      L     #HELP.WZ_rechts_3;
      L     #HELP.WZ_rechts_4;
      +R;
      T     #HELP.Sum_WZ_re_hinten;
      L     #HELP.AW_WZ_re_hinten;
      -R;
      ABS;
      L     #HELP.Tol_UeW_WZ;
      >R;
      A     #OUT.RUECK;
      S     #Kollision;

      A     #Kollision;
      A     #ZST.Unten_re;
      S     #ErrIn.Alarm.Koll_LF;

      A     #Kollision;
      A     #ZST.Oben_re;
      S     #ErrIn.Alarm.Koll_WF;


NETWORK
TITLE = allgemeine Fehlerbehandlung/Überwachungsfunktionen + Fehlerevent
// überwacht die Fahrwagenfunktionen in allen Betriebsarten
// ======== LASER ===========
Err:  L     S5T#5S;
      A     #ZST.AKTIV;
      O     #BA_Wxl;
      SF    T [#Timer3];

      A     T [#Timer3];
      O     #PAR.Free.Laser_req;
      O     "DB_ANLAGE".BA.Mess_on;
      =     #OUT.Req_Laser;

      L     S5T#1M;
      AN    #ZST.Auto;
      SD    T [#Timer0];
      A     "T_Verz_Auto";
      A     T [#Timer0];
      =     #MLD.Warnung.WARN_nAuto;

//--------------------------
//WT am TW nicht umsetzbar (FB9)
//--------------------------
      AN    #ZST.Auto;
      O     #ZST.Halt;
      ON    #ZST.BEREIT;
      O     #IN.QUITT_ALARM;
      O     #F_Taste;
      R     #ErrIn.Warnung.Wrn_WT_nUmsetzbar;

      A     #ErrIn.Warnung.Wrn_WT_nUmsetzbar;
      A     #ZST.Auto;
      =     #MLD.Warnung.WARN_WT_nUms;

//--------------------------
//FW-allgemein
//--------------------------
      A     #ErrIn.Alarm.F_Brk_Fahr;
      =     #MLD.Alarm_HW.F_Brk_Fahr;

//--------------------------
//Positioniersystem
//--------------------------
      AN    #ZST.REFERENZIERT;
      =     #MLD.Alarm_SW.nReferenz;

      A     #ErrIn.Alarm.PosSys;
      =     #MLD.Alarm_HW.PosSys;

      SET;
      R     #ErrPosSys;

      A     #ErrIn.Warnung.Wrn_Optik_PosSys;
      O     #ErrIn.Warnung.Wrn_Temp_PosSys;
      O     #ErrIn.Warnung.Wrn_Plaus_PosSys;
      JC    CNTp;

      L     0;
      T     #HELP.Count_PosSys;
      JU    eRRp;

CNTp: L     #HELP.Count_PosSys;
      L     30;
      >I;
      S     #ErrPosSys;
      JC    eRRp;
      AN    "Imp_1Hz";
      JC    eRRp;
      L     #HELP.Count_PosSys;
      +     1;
      T     #HELP.Count_PosSys;

eRRp: A     #ErrIn.Warnung.Wrn_Optik_PosSys;
      A     #ErrPosSys;
      =     #MLD.Warnung.Optik_PosSys;

      A     #ErrIn.Warnung.Wrn_Temp_PosSys;
      A     #ErrPosSys;
      =     #MLD.Warnung.Temp_PosSys;

      A     #ErrIn.Warnung.Wrn_Plaus_PosSys;
      A     #ErrPosSys;
      =     #MLD.Warnung.Wrn_Plaus_PosSys;

//Einschaltverzögerung Laser
      AN    #OUT.Req_Laser;
      O     #IN.Laser_on;
      L     0;
      JC    Loff;
      L     #HELP.Count_Laser_on;
      AN    "Imp_1Hz";
      JC    Loff;
      +     1;
Loff: T     #HELP.Count_Laser_on;

      L     #HELP.Count_Laser_on;
      L     5;
      >I;
      =     #MLD.Alarm_SW.Laser_off;

      A     #ErrIn.Warnung.Wrn_Temp_Fahr;
      A     #ZST.BEREIT;
      AN    #ErrIn.Alarm.Profinet_IO_nok;
      =     #MLD.Alarm_HW.Temp_Fahrt;
      A     #ErrIn.Warnung.Wrn_Temp_Fahr;
      AN    #ZST.BEREIT;
      AN    #ErrIn.Alarm.Profinet_IO_nok;
      =     #MLD.Warnung.Temp_Fahrt;
      A     #ErrIn.Alarm.Fahrt_nok;
      =     #MLD.Alarm_HW.St_FU_Fahrt;

      A     #ErrIn.Warnung.Wrn_Temp_Hub;
      A     #ZST.BEREIT;
      AN    #ErrIn.Alarm.Profinet_IO_nok;
      =     #MLD.Alarm_HW.Temp_Hub;

      A     #ErrIn.Warnung.Wrn_Temp_Hub;
      AN    #ZST.BEREIT;
      AN    #ErrIn.Alarm.Profinet_IO_nok;
      =     #MLD.Warnung.Temp_Hub;

//--------------------------
//Hubsystem
//--------------------------
      A     #ErrIn.Alarm.HubSys_li;
      =     #MLD.Alarm_HW.HubSys_li;

      A     #ErrIn.Alarm.HubSys_re;
      =     #MLD.Alarm_HW.HubSys_re;

      A     #ErrIn.Alarm.Hub_nok_links;
      =     #MLD.Alarm_HW.St_FU_Hub_li;
      A     #ErrIn.Alarm.Hub_nok_rechts;
      =     #MLD.Alarm_HW.St_FU_Hub_re;

      A     #ErrIn.Alarm.F_Brk_Hub_links;
      =     #MLD.Alarm_HW.F_Brk_Hub_li;
      A     #ErrIn.Alarm.F_Brk_Hub_rechts;
      =     #MLD.Alarm_HW.F_Brk_Hub_re;

//--------------------------
//Bereichs-/Kollisionsfehler
//--------------------------
      A     #ErrIn.Alarm.BE_Vor;
      AN    #ErrIn.Alarm.Profinet_IO_nok;
      =     #MLD.Alarm_HW.BE_vor;
      A     #ErrIn.Alarm.BE_Rck;
      AN    #ErrIn.Alarm.Profinet_IO_nok;
      =     #MLD.Alarm_HW.BE_rck;
      A     #ErrIn.Alarm.Gurt_UP_links;
      AN    #ErrIn.Alarm.Profinet_IO_nok;
      =     #MLD.Alarm_HW.GE_oben_li;
      A     #ErrIn.Alarm.Gurt_DN_links;
      AN    #ErrIn.Alarm.Profinet_IO_nok;
      =     #MLD.Alarm_HW.GE_unten_li;
      A     #ErrIn.Alarm.Gurt_UP_rechts;
      AN    #ErrIn.Alarm.Profinet_IO_nok;
      =     #MLD.Alarm_HW.GE_oben_re;
      A     #ErrIn.Alarm.Gurt_DN_rechts;
      AN    #ErrIn.Alarm.Profinet_IO_nok;
      =     #MLD.Alarm_HW.GE_unten_re;

      A     #ErrIn.Alarm.Koll_LF;
      AN    #ErrIn.Alarm.Profinet_IO_nok;
      S     #MLD.Alarm_HW.Koll_LF;
      A     #ErrIn.Alarm.Koll_WF;
      AN    #ErrIn.Alarm.Profinet_IO_nok;
      S     #MLD.Alarm_HW.Koll_WF;

      A     #ErrIn.Alarm.AFS_BS;
      AN    #ErrIn.Alarm.Profinet_IO_nok;
      =     #MLD.Alarm_HW.Afs_BS;
      A     #ErrIn.Alarm.AFS_WS;
      AN    #ErrIn.Alarm.Profinet_IO_nok;
      =     #MLD.Alarm_HW.Afs_WS;

      A     #ErrIn.Alarm.Last_UeW_links;
      =     #MLD.Alarm_HW.Last_UeW_li;

      A     #ErrIn.Alarm.Last_UeW_rechts;
      =     #MLD.Alarm_HW.Last_UeW_re;

      A     #ErrIn.Alarm.Gurt_UeL_links;
      AN    #ErrIn.Alarm.Profinet_IO_nok;
      =     #MLD.Alarm_HW.GurtUeL_li;

      A     #ErrIn.Alarm.Gurt_UeL_rechts;
      AN    #ErrIn.Alarm.Profinet_IO_nok;
      =     #MLD.Alarm_HW.GurtUeL_re;

      A     #ErrIn.Alarm.Profinet_IO_nok;
      =     #MLD.Alarm_HW.Profinet_nok;

//--------------------------
//Diagnose-/Fehlermeldung
//--------------------------
//:::::::::::::::::::::::::::::::
// Neustart AMS-alle Fehler neu
//:::::::::::::::::::::::::::::::
      AN    "DB_ANLAGE".IN.AMS_Restart;
      JC    NRes;
      L     0;
      T     #MLD.AM_ALHW;
      T     #MLD.AM_ALSW;
      T     #MLD.AM_WARN;
NRes: NOP   0;
//:::::::::::::::::::::::::::::::
// NotAus keine Fehlerbehandlung
//:::::::::::::::::::::::::::::::
      A     #ErrIn.Alarm.NotHalt;
      S     #ZST.FEHLER;
      JC    AOFF;
//:::::::::::::::::::::::::::::::
// Adresse initialisieren
//:::::::::::::::::::::::::::::::
      L     406;
      SLD   3;
      LAR1;
//:::::::::::::::::::::::::::::::
// Schleife über alle Fehler
//:::::::::::::::::::::::::::::::
      L     1;
reA:  T     #TMP.FHLR_NR;
      L     96;
      >I;
      JC    AEnd;
//:::::::::::::::::::::::::::::::
// Fehler gekommen/gegangen
//:::::::::::::::::::::::::::::::
      A     DIX [AR1, P#0.0];
      X     DIX [AR1, P#12.0];
      JCN   nxA;
      A     DIX [AR1, P#0.0];
      =     #new;

AOUT: NOP   0;

//:::::::::::::::::::::::::::::::
// Fehler neu--> Hupe
//:::::::::::::::::::::::::::::::
      A     #new;
      R     "DB_ANLAGE".config.M_Q_Hupe;

//:::::::::::::::::::::::::::::::
// nächster Fehler
//:::::::::::::::::::::::::::::::
nxA:  +AR1  P#0.1;
      L     #TMP.FHLR_NR;
      +     1;
      JU    reA;

//:::::::::::::::::::::::::::::::
// Altmerker Sichern
//:::::::::::::::::::::::::::::::
AEnd: L     %DID406;  //#MLD.Alarm_HW.xx
      T     #MLD.AM_ALHW;
      L     %DID410;  //#MLD.Alarm_SW.xx
      T     #MLD.AM_ALSW;
      L     %DID414;  //#MLD.Warnung.xx
      T     #MLD.AM_WARN;

//:::::::::::::::::::::::::::::::
// Fehlerzustand
//:::::::::::::::::::::::::::::::
      L     #MLD.AM_ALHW;
      L     0;
      <>D;
      O(;
      L     #MLD.AM_ALSW;
      <>D;
      );
      S     #ZST.FEHLER;

//:::::::::::::::::::::::::::::::::
// keine Fehler aber Fehlerzustand
//:::::::::::::::::::::::::::::::::
      L     %DID406;  //#MLD.Alarm_HW.xx
      L     0;
      ==D;
      A(;
      L     %DID410;  //#MLD.Alarm_SW.xx
      ==D;
      );
      A     #ZST.FEHLER;
      AN    #IN.QUITT_ALARM;
      S     #MLD.Alarm_SW.Fehler_Quitt;

      A     #ZST.FEHLER;
      AN    #ZST.Tipp;
      JC    AOFF;

      AN    #ZST.Halt;
      O     #ZST.Tipp;
      JC    WT;

//Alles Aus
AOFF: L     0;  //Ausgänge aus
      T     %DIW68;


NETWORK
TITLE = Warenträgerverwaltung
// kopiert WTs in und aus Positionen
// lädt Parameter usw.
WT:   L     #Adr_IstPos;
      LAR1;
      OPN   "DB_POS";
      L     #PAR.FW_Nr;
      T     DBB [AR1, P#5.0];  //FW_Nr im Bad ungerade
      T     DBB [AR1, P#105.0];  //FW_Nr im Bad gerade

      AN    #WTon_li;
      JC    nUms_li;
      L     #ZST.WT_DB_NR_li;
      +     100;
      T     #WT_DB_NR_li;

      OPN   DB [#WT_DB_NR_li];
      L     #PAR.FW_Nr;
      T     %DBB34;  //"DB_WT1".FW_Nr
nUms_li:A     #WTon_li;
      JC    WTaF_li;
      L     0;
      T     #ZST.Verweil;

WTaF_li:A     #ZST.low_SU_li;
      FN    #TMP.FM_low_SU_li;
      =     #FN_low_SU_li;

      AN    #ZST.Mittig;  //Umladen nur in PosMitte
      JC    WT_rechts;

//--------------------------------
//Kopieren WT in bzw. aus Pos
//--------------------------------
      A     #ZST.low_SU_li;
      A     #WTon_li;
      AN    #WT_in_Pos_li;
      A     #TMP.old_hub;  //#ZST.SENKEN_AKT
      JC    WT_P_li;
      A     #FN_low_SU_li;
      AN    #WTon_li;
      A     #WT_in_Pos_li;
      A     #TMP.old_hub;  //#ZST.HEBEN_AKT
      JC    WT_F_li;
      JU    WT_rechts;
//--------------------------------
//WT in Position laden
//--------------------------------
WT_P_li:L     #ZST.POSITION_li;
      T     #Nummer;

      CALL  "FC_WT_to_Pos"
      ( Pos_Nr     := #Nummer,
        WT_Nr      := #ZST.WT_DB_NR_li,
        BA_Auto    := #ZST.Auto,
        send_DBEvt := TRUE,
        SimLoad    := FALSE,
        Copy_ok    := #"Return"
      );

      AN    #"Return";
      JC    WT_rechts;
      R     #WTon_li;

      L     0;  //löschen am FW
      T     #ZST.WT_DB_NR_li;
      T     #ZST.WT_NR_LANG_li;
      JU    WT_rechts;

//--------------------------------
//WT aus Position laden
//--------------------------------
WT_F_li:L     #ZST.POSITION_li;
      T     #Nummer;

      CALL  "FC_WT_from_Pos"
      ( Pos_Nr     := #Nummer,
        send_DBEvt := TRUE,
        load_ok    := #"Return",
        WT_Nr      := #ZST.WT_DB_NR_li,
        WT_Nr_lang := #ZST.WT_NR_LANG_li
      );

      AN    #"Return";
      JC    WT_rechts;
      S     #WTon_li;

      AN    #ZST.Auto;
      JC    WT_rechts;

      L     #ZST.WT_DB_NR_li;
      +     100;
      T     #WT_DB_NR_li;

      OPN   DB [#WT_DB_NR_li];
      L     %DBB36;  //WT-Ziel bereits festgelegt
      L     0;
      <>I;
      JC    Zset_li;
      L     %DBB21;
      T     %DBB36;  //WT-Ziel

Zset_li:L     #TMP.ZielPos;
      T     %DBB21;

      L     #TMP.ZielPos;
      T     #Nummer;
      CALL  "FC_WT_to_Pos"
      ( Pos_Nr     := #Nummer,
        WT_Nr      := #ZST.WT_DB_NR_li,
        BA_Auto    := #ZST.Auto,
        send_DBEvt := FALSE,
        SimLoad    := TRUE,
        Copy_ok    := #"Return"
      );

WT_rechts:NOP   0;

      AN    #WTon_re;
      JC    nUms_re;
      L     #ZST.WT_DB_NR_re;
      +     100;
      T     #WT_DB_NR_re;

      OPN   DB [#WT_DB_NR_re];
      L     #PAR.FW_Nr;
      T     %DBB34;  //"DB_WT1".FW_Nr
nUms_re:A     #WTon_re;
      JC    WTaF_re;
      L     0;
      T     #ZST.Verweil;

WTaF_re:A     #ZST.low_SU_re;
      FN    #TMP.FM_low_SU_re;
      =     #FN_low_SU_re;

      AN    #ZST.Mittig;  //Umladen nur in PosMitte
      JC    Komm;

//--------------------------------
//Kopieren WT in bzw. aus Pos
//--------------------------------
      A     #ZST.low_SU_re;
      A     #WTon_re;
      AN    #WT_in_Pos_re;
      A     #TMP.old_hub;  //#ZST.SENKEN_AKT
      JC    WT_P_re;
      A     #FN_low_SU_re;
      AN    #WTon_re;
      A     #WT_in_Pos_re;
      A     #TMP.old_hub;  //#ZST.HEBEN_AKT
      JC    WT_F_re;
      JU    Komm;
//--------------------------------
//WT in Position laden
//--------------------------------
WT_P_re:L     #ZST.POSITION_re;
      T     #Nummer;

      CALL  "FC_WT_to_Pos"
      ( Pos_Nr     := #Nummer,
        WT_Nr      := #ZST.WT_DB_NR_re,
        BA_Auto    := #ZST.Auto,
        send_DBEvt := TRUE,
        SimLoad    := FALSE,
        Copy_ok    := #"Return"
      );

      AN    #"Return";
      JC    Komm;
      R     #WTon_re;

      L     0;  //löschen am FW
      T     #ZST.WT_DB_NR_re;
      T     #HELP.WT_NR_LANG_re;
      JU    Komm;

//--------------------------------
//WT aus Position laden
//--------------------------------
WT_F_re:L     #ZST.POSITION_re;
      T     #Nummer;

      CALL  "FC_WT_from_Pos"
      ( Pos_Nr     := #Nummer,
        send_DBEvt := TRUE,
        load_ok    := #"Return",
        WT_Nr      := #ZST.WT_DB_NR_re,
        WT_Nr_lang := #HELP.WT_NR_LANG_re
      );

      AN    #"Return";
      JC    Komm;
      S     #WTon_re;

      AN    #ZST.Auto;
      JC    Komm;

      L     #ZST.WT_DB_NR_re;
      +     100;
      T     #WT_DB_NR_re;

      OPN   DB [#WT_DB_NR_re];
      L     %DBB36;  //WT-Ziel bereits festgelegt
      L     0;
      <>I;
      JC    Zset_re;
      L     %DBB21;
      T     %DBB36;  //WT-Ziel

Zset_re:L     #TMP.ZielPos;
      T     %DBB21;

      L     #TMP.ZielPos;
      T     #Nummer;
      CALL  "FC_WT_to_Pos"
      ( Pos_Nr     := #Nummer,
        WT_Nr      := #ZST.WT_DB_NR_re,
        BA_Auto    := #ZST.Auto,
        send_DBEvt := FALSE,
        SimLoad    := TRUE,
        Copy_ok    := #"Return"
      );


NETWORK
TITLE = Kommunikation zu Partnerfunktionen
// Datenübertragung zu PC, Optimierung, Diagwatch usw.
// Ziel-Quelle-Informationen, Heben-Senken-Informationen in Positionen anmelden
Komm: NOP   0;
//---------------------------
//Positionsinformationen DB51
//---------------------------
      L     #Adr_IstPos;
      LAR1;
      OPN   "DB_POS";
      A     #ZST.HEBEN_AKT;  // #OUT.HEBEN
      =     DBX [AR1, P#6.6];  //FW Heben
      =     DBX [AR1, P#106.6];  //FW Heben
      A     #ZST.SENKEN_AKT;  // #OUT.SENKEN
      =     DBX [AR1, P#6.7];  //FW Senken
      =     DBX [AR1, P#106.7];  //FW Senken

      AN    #ZST.VORWAERTS_AKT;
      AN    #ZST.RUECKWAERTS_AKT;
      A     #ZST.Mittig;
      =     DBX [AR1, P#6.5];  //FW in Pos
      =     DBX [AR1, P#106.5];  //FW in Pos

//FW-kommt in allen Positionen setzen,die überfahren werden
      L     0;
      L     #TMP.ZielPos;
      ==I;
      JC    noZ;
      L     2;
      MOD;
      L     #TMP.ZielPos;
      JP    linke_S;
      DEC   1;
linke_S:L     #ZST.POSITION_li;
      <I;
      JC    ldC;
      CAC;
ldC:  T     #PCount_hi;
      CAC;
retC: T     #PCount_low;
      L     "DB_POS".LENG;
      *I;
      L     "DB_POS".Offset;
      +I;
      SLD   3;
      LAR1;
      OPN   "DB_POS";
      S     DBX [AR1, P#6.4];  //FW kommt
      S     DBX [AR1, P#106.4];  //FW kommt
      L     #PCount_hi;
      L     #PCount_low;
      <=I;
      JC    noZ;
      +     2;
      JU    retC;

noZ:  AN    #ZST.Auto;
      JC    noto;
      L     %DIB31;  //Befehlsart
      L     16#03;
      <>I;
      JC    noto;
//Ziel sperren
      L     0;
      L     %DIB33;
      ==I;
      JC    noto;
      L     "DB_POS".LENG;
      *I;
      L     "DB_POS".Offset;
      +I;
      SLD   3;
      LAR1;
      OPN   "DB_POS";
      S     DBX [AR1, P#6.3];  //reserviertes Ziel
      AN    #WTon_li;
      AN    #WTon_re;
      JC    Qset;

      AN    #WTon_li;
      JC    rZ_re;
      L     #ZST.WT_DB_NR_li;
      T     DBB [AR1, P#36.0];  //Next-WT

      AN    #WTon_re;
      JC    Qset;
      L     #ZST.WT_DB_NR_re;
      T     DBB [AR1, P#136.0];  //Next-WT
      JU    Qset;

rZ_re:AN    #WTon_re;
      JC    Qset;
      L     #ZST.WT_DB_NR_re;
      T     DBB [AR1, P#36.0];  //Next-WT

//Quelle sperren
Qset: A     #WTon_li;
      O     #WTon_re;
      JC    noto;
      L     0;
      L     %DIB32;
      ==I;
      JC    noto;
      L     "DB_POS".LENG;
      *I;
      L     "DB_POS".Offset;
      +I;
      SLD   3;
      LAR1;
      OPN   "DB_POS";
      S     DBX [AR1, P#6.2];  //reservierte Quelle

noto: BE;

END_FUNCTION_BLOCK

FUNCTION "FC_Pos_Erk" : Void   // FC11, STL
TITLE = Positioniersystem
{ S7_Optimized_Access := 'FALSE' }
AUTHOR : MS
FAMILY : FW
// stored: AutoNumber false
   VAR_INPUT
      Instanz_DB : Int;
   END_VAR
   VAR_TEMP
      FW_DB : DB_ANY;
      Abstand : DInt;
      Pos : Byte;
      count : Byte;
      rotWert : Word;
      frstChk : Bool;
      minGrenze : Byte;
      maxGrenze : Byte;
      Grenze_min : DInt;
      Grenze_max : DInt;
      SU_Ebene_0 : DInt;
   END_VAR
BEGIN

NETWORK
TITLE = Position ermitteln
// Inkrementwert wird auf minimalen Abstand einer Positionsmitte überprüft.
// Position mit geringstem Abstand wird übernommen.
      L     #Instanz_DB;
      T     #FW_DB;
      OPN   DI [#FW_DB];

      SET;
      =     #frstChk;
      L     0;
      T     #SU_Ebene_0;

      L     "DI_FW_1".PAR.Fahrt.FAHRBEREICH_MIN;
      T     #minGrenze;
      L     "DI_FW_1".PAR.Fahrt.FAHRBEREICH_MAX;
      T     #maxGrenze;
      L     "DI_FW_1".IN.Grenze_min;
      T     #Grenze_min;
      L     "DI_FW_1".IN.Grenze_max;
      T     #Grenze_max;

      L     "DI_FW_1".PAR.Fahrt.FAHRBEREICH_MIN;
      T     #Pos;
retP: T     #count;
      L     "DI_FW_1".PAR.Fahrt.FAHRBEREICH_MAX;
      +     -1;  // HCA: nur ungerade Pos. zählen
      >I;
      JC    ckok;

      L     #count;
      L     "DB_POS".LENG;
      *D;
      L     "DB_POS".Offset;
      +D;
      SLD   3;
      LAR1;
      OPN   "DB_POS";
      L     #Grenze_min;
      L     DBD [AR1, P#22.0];  //BadPos in Inc
      <=D;
      JC    gmin;
      L     #count;
      +     2;  // HCA: nur ungeradePos. zählen
      T     #minGrenze;
gmin: L     #Grenze_max;
      OPN   "DB_POS";
      L     DBD [AR1, P#22.0];  //BadPos in Inc
      <D;
      JC    gmax;
      L     #count;
      T     #maxGrenze;
gmax: NOP   0;
      OPN   "DB_POS";
      L     DBD [AR1, P#22.0];  //BadPos in Inc
      L     "DI_FW_1".ZST.PosInc;
      -D;
      DTR;
      ABS;
      RND;
      L     #Abstand;
      >=D;
      AN    #frstChk;
      JC    nexP;
      R     #frstChk;
      CAC;
      T     #Abstand;
      L     #count;
      T     #Pos;

nexP: L     #count;
      L     2;  // HCA: nur ungeradePos. zählen
      +I;
      JU    retP;

ckok: L     #Pos;
      T     "DI_FW_1".ZST.POSITION_li;

      L     #Abstand;
      L     "DI_FW_1".PAR.Fahrt.Bereich_Pos;
      <=D;
      =     "DI_FW_1".ZST.Mittig;

// Ofs-Mittig
      L     #Pos;
      L     "DB_POS".LENG;
      *D;
      L     "DB_POS".Offset;
      +D;
      SLD   3;
      LAR1;
      OPN   "DB_POS";
      L     DBD [AR1, P#22.0];  //BadPos in Inc
      L     DBD [AR1, P#64.0];  //"DB_POS".POS[x].SonderPos_Offset
      -D;
      L     "DI_FW_1".ZST.PosInc;
      -D;
      DTR;
      ABS;
      RND;
      L     "DI_FW_1".PAR.Fahrt.Bereich_Pos;
      <=D;
      =     "DI_FW_1".ZST.Ofs_mittig;

// Tiefsenkbereich
      A(;
      OPN   "DB_POS";
      L     DBD [AR1, P#22.0];  //Posmitte
      L     "DI_FW_1".PAR.Fahrt.Bereich_Pos;
      +D;
      L     "DI_FW_1".ZST.PosInc;
      >D;
      );
      A(;
      OPN   "DB_POS";
      L     DBD [AR1, P#22.0];  //Posmitte
      L     DBD [AR1, P#64.0];  //"DB_POS".POS[x].SonderPos_Offset
      -D;
      L     "DI_FW_1".PAR.Fahrt.Bereich_Pos;
      -D;
      L     "DI_FW_1".ZST.PosInc;
      <D;
      );
      A(;
      A     "DI_FW_1".IN.Unten_li;
      O     "DI_FW_1".IN.Unten_re;
      );
      =     "DI_FW_1".ZST.Ofs_Bereich;

// Absetzhöhe
      OPN   "DB_POS";
      L     0;
      L     DBD [AR1, P#14.0];  //"DB_POS".POS[x].Absetzhoehe
      >=D;
      JC    VZB;
      T     "DI_FW_1".PAR.Hub.Ebene0;

//Vorzugsbereich min ungültig?
VZB:  L     "DI_FW_1".PAR.Fahrt.FAHRBEREICH_MIN;
      L     "DI_FW_1".PAR.Vorzugsbereich_max;
      >I;
      O(;
      L     "DI_FW_1".PAR.Fahrt.FAHRBEREICH_MAX;
      >I;
      );
      JC    Gclr;
//ggf. Korrektur min
      L     #maxGrenze;
      L     "DI_FW_1".PAR.Vorzugsbereich_max;
      <=I;
      JC    Gclr;
      T     #minGrenze;
Gclr: NOP   0;

//Vorzugsbereich min ungültig?
      L     "DI_FW_1".PAR.Fahrt.FAHRBEREICH_MIN;
      L     "DI_FW_1".PAR.Vorzugsbereich_min;
      >I;
      O(;
      L     "DI_FW_1".PAR.Fahrt.FAHRBEREICH_MAX;
      >I;
      );
      JC    Gset;
//ggf. Korrektur min
      L     #minGrenze;
      L     "DI_FW_1".PAR.Vorzugsbereich_min;
      >=I;
      JC    Gset;
      T     #minGrenze;

Gset: L     #minGrenze;
      T     "DI_FW_1".HELP.Grenze_min;
      L     #maxGrenze;
      T     "DI_FW_1".HELP.Grenze_max;




NETWORK
TITLE = nächsten HW ermitteln
ChHW: NOP   0;
      AN    "DB_ANLAGE".config.HW_exist;
      R     "DI_FW_1".ZST.HW_mittig;
      L     1;  //temp. Hubeben
      JC    SUok;

      SET;
      =     #frstChk;

      L     0;
      T     #Pos;
retH: T     #count;
      L     "DB_HW".Anzahl;
      >=I;
      JC    Hok;

      L     #count;
      L     "DB_HW".lengHW;
      *D;
      L     "DB_HW".Offset;
      +D;
      SLD   3;
      LAR1;
      OPN   "DB_HW";
      L     0;
      L     DBD [AR1, P#0.0];  //HW-Pos in Inc
      ==D;
      JC    Hok;
      L     "DI_FW_1".ZST.PosInc;
      -D;
      DTR;
      ABS;
      RND;
      L     #Abstand;
      >=D;
      AN    #frstChk;
      JC    nexH;
      R     #frstChk;
      CAC;
      T     #Abstand;
      L     #count;
      T     #Pos;

nexH: L     #count;
      L     1;
      +I;
      JU    retH;

Hok:  L     #Abstand;
      L     "DI_FW_1".PAR.Fahrt.Bereich_Pos;
      <=D;
      =     "DI_FW_1".ZST.HW_mittig;


NETWORK
TITLE = aktuelle SU-Ebene ermitteln
      L     #Pos;
      L     "DB_HW".lengHW;
      *D;
      L     "DB_HW".Offset;
      +D;
      SLD   3;
      LAR1;
      A     "DI_FW_1".ZST.HW_mittig;
      JC    mitt;
      OPN   "DB_HW";
      L     DBD [AR1, P#0.0];  //HW-Pos in Inc
      L     "DI_FW_1".ZST.PosInc;
      -D;
      JP    vorH;
//FW ist hinter HW-Pos
      OPN   "DB_HW";
      L     DBB [AR1, P#5.0];  //HW-Ebene bei verlassen in Richtung vorwärts
      T     "DI_FW_1".TMP.low_SU_Ebene;
      L     1;
      SLW;  //Bit0==TRUE wird um Ebene verschoben
      JU    SUok;

//FW ist vor HW-Pos
vorH: OPN   "DB_HW";
      L     DBB [AR1, P#4.0];  //HW-Ebene bei verlassen in Richtung rückwärts
      T     "DI_FW_1".TMP.low_SU_Ebene;
      L     1;
      SLW;  //Bit0==TRUE wird um Ebene verschoben
      JU    SUok;

//FW ist auf HW-Pos
mitt: OPN   "DB_HW";
      L     DBB [AR1, P#4.0];  //HW-Ebene bei verlassen in Richtung rückwärts
      L     DBB [AR1, P#5.0];  //HW-Ebene bei verlassen in Richtung vorwärts
      >I;
      JC    lSU;
      CAC;
lSU:  T     "DI_FW_1".TMP.low_SU_Ebene;
      OPN   "DB_HW";
      L     DBB [AR1, P#4.0];  //HW-Ebene bei verlassen in Richtung rückwärts
      L     1;
      SLW;  //Bit0==TRUE wird um Ebene verschoben
      T     #rotWert;
      L     DBB [AR1, P#5.0];  //HW-Ebene bei verlassen in Richtung vorwärts
      L     1;
      SLW;  //Bit0==TRUE wird um Ebene verschoben
      L     #rotWert;
      OW;  //beide Ebenen gelten

SUok: T     "DI_FW_1".TMP.Hub_Ebenen;

      L     "DI_FW_1".TMP.low_SU_Ebene;
      T     "DI_FW_1".PAR.Hub.SUF_Ebene;

      A     "DI_FW_1".ZST.Mittig;
      O     "DI_FW_1".ZST.Ofs_Bereich;
      O     "DI_FW_1".ZST.Ofs_mittig;
      JCN   Z_E;
      L     0;
      T     "DI_FW_1".TMP.low_SU_Ebene;  // ganz unten erlaubt
      L     "DI_FW_1".TMP.Hub_Ebenen;
      OW    W#16#01;
      T     "DI_FW_1".TMP.Hub_Ebenen;

//SO- und Z-Ebene übergeben
Z_E:  L     0;
      L     "DI_FW_1".PAR.Hub.Z_Ebene;
      ==I;
      JC    SO;
      L     1;
      SLW;
      L     "DI_FW_1".TMP.Hub_Ebenen;
      OW;
      T     "DI_FW_1".TMP.Hub_Ebenen;
SO:   L     0;
      L     "DI_FW_1".PAR.Hub.SO_Ebene;
      ==I;
      BEC;
      L     1;
      SLW;
      L     "DI_FW_1".TMP.Hub_Ebenen;
      OW;
      T     "DI_FW_1".TMP.Hub_Ebenen;

END_FUNCTION

FUNCTION "FC_Hub_Erk_li" : Void   // FC12, STL
TITLE = Hubsystem
{ S7_Optimized_Access := 'FALSE' }
AUTHOR : MS
FAMILY : FW
// stored: AutoNumber false
   VAR_INPUT
      Instanz_DB : Int;
   END_VAR
   VAR_TEMP
      FW_DB : DB_ANY;
      Abstand : DInt;
      Ebene : Byte;
      count : Byte;
      rotWert : Word;
      frstChk : Bool;
   END_VAR
BEGIN

NETWORK
TITLE = Fahrwagen-Ebene ermitteln
// Inkrementwert wird auf minimalen Abstand zu einer Hubebene überprüft.
// Ebene mit geringstem Abstand wird übernommen.
      L     #Instanz_DB;
      T     #FW_DB;
      OPN   DI [#FW_DB];

      SET;
      =     #frstChk;

      L     0;
      T     #Ebene;
      T     #Abstand;
retE: T     #count;
      L     6;
      >I;
      JC    ckok;

      CAC;
      L     4;
      *D;
      L     292;
      +D;
      SLD   3;
      LAR1;

      L     0;
      L     DID [AR1, P#0.0];  //"DI_FW_1".PAR.Hub.Ebene...
      ==D;
      JC    ckok;
      L     "DI_FW_1".ZST.HubInc_li;
      -D;
      DTR;
      ABS;
      RND;
      L     #Abstand;
      >=D;
      AN    #frstChk;
      JC    nexE;
      R     #frstChk;
      CAC;
      T     #Abstand;
      L     #count;
      T     #Ebene;

nexE: L     #count;
      L     1;
      +I;
      JU    retE;

ckok: L     320;  //prüfen auf Z-Ebene
      SLD   3;
      LAR1;
      L     0;
      L     DID [AR1, P#0.0];  //"DI_FW_1".PAR.Hub.Ebene...
      ==D;
      JC    noZ;
      L     "DI_FW_1".ZST.HubInc_li;
      -D;
      DTR;
      ABS;
      RND;
      L     #Abstand;
      >=D;
      JC    noZ;
      CAC;
      T     #Abstand;
      L     7;
      T     #Ebene;

noZ:  L     #Ebene;
      T     "DI_FW_1".ZST.Ebene_li;

      L     #Abstand;
      L     "DI_FW_1".PAR.Hub.Bereich_Pos;
      <=D;
      AN    #frstChk;
      =     "DI_FW_1".ZST.HubSensor_li;


NETWORK
TITLE = SU/SO/Z setzen

      L     #Ebene;
      L     1;
      SLW;
      L     "DI_FW_1".PAR.Hub.SU_Ebenen;
      AW;
      L     "DI_FW_1".TMP.Hub_Ebenen;
      AW;
      L     0;
      <>I;
      A     "DI_FW_1".ZST.HubSensor_li;
      =     "DI_FW_1".ZST.Unten_li;

      L     #Ebene;
      L     "DI_FW_1".PAR.Hub.Z_Ebene;
      ==I;
      A     "DI_FW_1".ZST.HubSensor_li;
      =     "DI_FW_1".ZST.Z_Sensor_li;

      L     #Ebene;
      L     "DI_FW_1".PAR.Hub.SO_Ebene;
      ==I;
      A     "DI_FW_1".ZST.HubSensor_li;
      =     "DI_FW_1".ZST.Oben_li;

      L     #Ebene;
      L     0;
      ==I;
      R     "DI_FW_1".ZST.Z_Sensor_li;
      R     "DI_FW_1".ZST.Oben_li;

      A     "DI_FW_1".IN.Oben_li;
      S     "DI_FW_1".ZST.Oben_li;


NETWORK
TITLE = WT Kopierfreigabe
      L     "DI_FW_1".TMP.low_SU_Ebene;
      L     #Ebene;
      ==I;
      A     "DI_FW_1".ZST.HubSensor_li;
      =     "DI_FW_1".ZST.low_SU_li;

END_FUNCTION

FUNCTION "FC_Hub_Erk_re" : Void   // FC112, STL
TITLE = Hubsystem
{ S7_Optimized_Access := 'FALSE' }
AUTHOR : MS
FAMILY : FW
// stored: AutoNumber false
   VAR_INPUT
      Instanz_DB : Int;
   END_VAR
   VAR_TEMP
      FW_DB : DB_ANY;
      Abstand : DInt;
      Ebene : Byte;
      count : Byte;
      rotWert : Word;
      frstChk : Bool;
   END_VAR
BEGIN

NETWORK
TITLE = Fahrwagen-Ebene ermitteln
// Inkrementwert wird auf minimalen Abstand zu einer Hubebene überprüft.
// Ebene mit geringstem Abstand wird übernommen.
      L     #Instanz_DB;
      T     #FW_DB;
      OPN   DI [#FW_DB];

      SET;
      =     #frstChk;

      L     0;
      T     #Ebene;
      T     #Abstand;
retE: T     #count;
      L     6;
      >I;
      JC    ckok;

      CAC;
      L     4;
      *D;
      L     292;
      +D;
      SLD   3;
      LAR1;

      L     0;
      L     DID [AR1, P#0.0];  //"DI_FW_1".PAR.Hub.Ebene...
      ==D;
      JC    ckok;
      L     "DI_FW_1".HELP.HubInc_re;
      -D;
      DTR;
      ABS;
      RND;
      L     #Abstand;
      >=D;
      AN    #frstChk;
      JC    nexE;
      R     #frstChk;
      CAC;
      T     #Abstand;
      L     #count;
      T     #Ebene;

nexE: L     #count;
      L     1;
      +I;
      JU    retE;

ckok: L     320;  //prüfen auf Z-Ebene
      SLD   3;
      LAR1;
      L     0;
      L     DID [AR1, P#0.0];  //"DI_FW_1".PAR.Hub.Ebene...
      ==D;
      JC    noZ;
      L     "DI_FW_1".HELP.HubInc_re;
      -D;
      DTR;
      ABS;
      RND;
      L     #Abstand;
      >=D;
      JC    noZ;
      CAC;
      T     #Abstand;
      L     7;
      T     #Ebene;

noZ:  L     #Ebene;
      T     "DI_FW_1".ZST.Ebene_re;

      L     #Abstand;
      L     "DI_FW_1".PAR.Hub.Bereich_Pos;
      <=D;
      AN    #frstChk;
      =     "DI_FW_1".ZST.HubSensor_re;


NETWORK
TITLE = SU/SO/Z setzen

      L     #Ebene;
      L     1;
      SLW;
      L     "DI_FW_1".PAR.Hub.SU_Ebenen;
      AW;
      L     "DI_FW_1".TMP.Hub_Ebenen;
      AW;
      L     0;
      <>I;
      A     "DI_FW_1".ZST.HubSensor_re;
      =     "DI_FW_1".ZST.Unten_re;

      L     #Ebene;
      L     "DI_FW_1".PAR.Hub.Z_Ebene;
      ==I;
      A     "DI_FW_1".ZST.HubSensor_re;
      =     "DI_FW_1".ZST.Z_Sensor_re;

      L     #Ebene;
      L     "DI_FW_1".PAR.Hub.SO_Ebene;
      ==I;
      A     "DI_FW_1".ZST.HubSensor_re;
      =     "DI_FW_1".ZST.Oben_re;

      L     #Ebene;
      L     0;
      ==I;
      R     "DI_FW_1".ZST.Z_Sensor_re;
      R     "DI_FW_1".ZST.Oben_re;

      A     "DI_FW_1".IN.Oben_re;
      S     "DI_FW_1".ZST.Oben_re;


NETWORK
TITLE = WT Kopierfreigabe
      L     "DI_FW_1".TMP.low_SU_Ebene;
      L     #Ebene;
      ==I;
      A     "DI_FW_1".ZST.HubSensor_re;
      =     "DI_FW_1".ZST.low_SU_re;

END_FUNCTION

FUNCTION "FC_Transzeit" : Void   // FC35, STL
{ S7_Optimized_Access := 'FALSE' }
AUTHOR : MS
// stored: AutoNumber false
   VAR_INPUT
      Pos : Byte;
      Quelle : Byte;
      Ziel : Byte;
      FW_Nr : Byte;
      ChkLeerfahrt : Bool;   // nur Leerfahrt berechnen
      StartPos : Bool;   // inc. der Pos als Startposition
      KorrTime : DInt;   // Korrektur Zeit in der Zukunft
   END_VAR
   VAR_OUTPUT
      Fahrzeit : DInt;
   END_VAR
   VAR_TEMP
      Leerfahrt : Real;
      Hubzeit : Real;
      Tropfzeit : Real;
      Warenfahrt : Real;
      Pendelzeit : Real;
      Senkzeit : Real;
      Tropfwanne : Real;
      KorrAtz : Real;
      KorrPend : Real;
      Trommel : Bool;
      lngsm_h : Bool;
      lngsm_s : Bool;
      FWok : Bool;
      immer_schnell : Bool;
      TS_Pos : Bool;
      WT_DB : Int;
      savAr1 : DWord;
      FW_DB : Int;
      Abstand : Real;
      ProzSpeed : Real;
      Quellpos : DInt;
      Restzeit : DInt;
      IstInc : DInt;
   END_VAR
BEGIN

NETWORK
TITLE = Register retten
// --------------------------------
// Register retten
// --------------------------------
      TAR1;
      T     #savAr1;


NETWORK
TITLE = Init
      L     0;
      T     #Fahrzeit;
      T     #Leerfahrt;
      T     #Hubzeit;
      T     #Tropfzeit;
      T     #Warenfahrt;
      T     #Pendelzeit;
      T     #Senkzeit;
      T     #Tropfwanne;

      SET;
      =     #TS_Pos;

      L     #FW_Nr;
      L     0;
      >I;
      =     #FWok;

      L     #FW_Nr;
      L     "DB_ANLAGE".config.ANZ_FW;
      >I;
      R     #FWok;
      R     #TS_Pos;

      L     1;
      L     #Quelle;
      >I;
      O(;
      L     "DB_ANLAGE".config.ANZ_Pos;
      >I;
      );
      JC    raus;

      A     #ChkLeerfahrt;
      JC    Leer;

      L     1;
      L     #Ziel;
      >I;
      O(;
      L     "DB_ANLAGE".config.ANZ_Pos;
      >I;
      );
      JC    raus;

Leer: NOP   0;

NETWORK
TITLE = Leerfahrt
      L     #Pos;
      L     "DB_POS".LENG;
      *D;
      L     "DB_POS".Offset;
      +D;
      SLD   3;
      LAR1;
      OPN   "DB_POS";
      L     DBD [AR1, P#22.0];  //"DB_POS".POS[0].IncPos
      T     #IstInc;

      L     #Quelle;
      L     "DB_POS".LENG;
      *D;
      L     "DB_POS".Offset;
      +D;
      SLD   3;
      LAR1;
      OPN   "DB_POS";
      AN    DBX [AR1, P#8.0];  //"DB_POS".POS[0].TS_Pos
      R     #TS_Pos;
      A     DBX [AR1, P#10.2];  //"DB_POS".POS[0].ignor_Exp
      L     0;
      JC    okRT;
      L     DBD [AR1, P#60.0];  //"DB_POS".POS[0].Korr_Restzeit
      L     #KorrTime;
      -D;
      JP    okRT;
      L     0;
okRT: DTR;
      T     #Restzeit;

      A     #FWok;
      A     "DB_ANLAGE".config.Pos_absolut;
      JC    LFa;

//Leerfahrzeit Sensor berechnen
      L     #Pos;
      L     #Quelle;
      -I;
      ITD;
      DTR;
      ABS;
      L     0.0;
      ==R;
      JC    LF;
      CAC;
      L     1.0;
      -R;
      L     "DB_Fahr-Hubzeit".FZ_Typ_Pos;
      *R;
      L     "DB_Fahr-Hubzeit".FZ_Typ_Halt;
      +R;
      JU    LF;

//Leerfahrzeit absolut berechnen
LFa:  L     #Quelle;
      L     "DB_POS".LENG;
      *D;
      L     "DB_POS".Offset;
      +D;
      SLD   3;
      LAR1;
      OPN   "DB_POS";
      L     DBD [AR1, P#22.0];  //"DB_POS".POS[0].IncPos
      T     #Quellpos;
      L     DBB [AR1, P#36.0];  //WT-DB
      +     100;
      T     #WT_DB;

      L     #FW_Nr;
      +     10;
      T     #FW_DB;

      A     #StartPos;
      L     #IstInc;
      JC    EPQ;

      OPN   DB [#FW_DB];
      L     0;
      L     %DBW366;  //"DI_FW_1".TMP.EndZiel
      ==I;
      JC    rdyQ;
      L     "DB_POS".LENG;
      *D;
      L     "DB_POS".Offset;
      +D;
      SLD   3;
      LAR1;
      OPN   "DB_POS";
      L     DBD [AR1, P#22.0];  //"DB_POS".POS[0].IncPos
      JU    EPQ;

rdyQ: OPN   DB [#FW_DB];
      L     %DBD4;  //"DI_FW_1".ZST.PosInc
EPQ:  L     #Quellpos;
      -D;
      DTR;
      ABS;
      T     #Abstand;
      L     0.0;
      ==D;
      JC    LF;

      OPN   DB [#FW_DB];
      L     %DBW246;  //"DI_FW_1".PAR.Fahrt.Fahr_DBNr
      T     #FW_DB;
      OPN   DB [#FW_DB];
      L     %DBW12;  //"DI_FW_POS_1".Config.Speed.Max
      ITD;
      DTR;
      L     100.0;
      /R;
      T     #ProzSpeed;

      L     %DBD22;  //"DI_FW_POS_1".Config.Rampe.Auf_Leer
      L     %DBD26;  //"DI_FW_POS_1".Config.Rampe.Ab_Leer
      +R;
      L     2.0;
      /R;
      L     #ProzSpeed;
      *R;
      T     #Leerfahrt;  //Zeit für Rampen
      L     %DBD14;  //"DI_FW_POS_1".Config.Speed.Norm mm/s
      *R;
      L     2.0;
      /R;
      L     #Abstand;
      CAC;
      -R;
      T     #Abstand;  //Weg für Konstantfahrt
      L     0.0;
      <=R;
      JC    endL;

      L     %DBD14;  //"DI_FW_POS_1".Config.Speed.Norm mm/s
      L     #ProzSpeed;
      *R;
      L     #Abstand;
      CAC;
      /R;
      L     #Leerfahrt;
      +R;
LF:   T     #Leerfahrt;
endL: SET;
      A     #ChkLeerfahrt;
      JC    Zeit;

NETWORK
TITLE = Warenfahrt
      L     #Quelle;
      L     #Ziel;
      -I;
      ITD;
      DTR;
      ABS;
      L     0.0;
      ==R;
      JC    WF;

      A     #FWok;
      A     "DB_ANLAGE".config.Pos_absolut;
      JC    WFa;
//Warenfahrzeit Sensor berechnen
      CAC;
      L     1.0;
      -R;
      L     "DB_Fahr-Hubzeit".FZ_Typ_Pos;
      *R;
      L     "DB_Fahr-Hubzeit".FZ_Typ_Halt;
      +R;
      JU    WF;

//Warenfahrzeit absolut berechnen
WFa:  L     #Ziel;
      L     "DB_POS".LENG;
      *D;
      L     "DB_POS".Offset;
      +D;
      SLD   3;
      LAR1;
      OPN   "DB_POS";
      L     DBD [AR1, P#22.0];  //"DB_POS".POS[0].IncPos
      L     #Quellpos;
      -D;
      DTR;
      ABS;
      T     #Abstand;
      L     0.0;
      ==D;
      JC    WF;

      L     1.0;
      T     #ProzSpeed;

      L     100;
      L     #WT_DB;
      >=I;
      JC    nWT;
      OPN   DB [#WT_DB];
      L     %DBW68;  //"DB_WT1".Speed_Fahrt
      ITD;
      DTR;
      L     100.0;
      /R;
      T     #ProzSpeed;

nWT:  L     #FW_Nr;
      +     10;
      T     #FW_DB;

      OPN   DB [#FW_DB];
      AN    %DBX343.0;  //"DI_FW_1".PAR.Free.TS
      R     #TS_Pos;
      L     %DBW246;  //"DI_FW_1".PAR.Fahrt.Fahr_DBNr
      T     #FW_DB;
      OPN   DB [#FW_DB];
      L     %DBW12;  //"DI_FW_POS_1".Config.Speed.Max
      ITD;
      DTR;
      L     100.0;
      /R;
      L     #ProzSpeed;
      *R;
      T     #ProzSpeed;

      L     %DBD30;  //"DI_FW_POS_1".Config.Rampe.Auf_Ware
      L     %DBD34;  //"DI_FW_POS_1".Config.Rampe.Ab_Ware
      +R;
      L     2.0;
      /R;
      L     #ProzSpeed;
      *R;
      T     #Warenfahrt;  //Zeit für Rampen
      L     %DBD14;  //"DI_FW_POS_1".Config.Speed.Norm mm/s
      *R;
      L     2.0;
      /R;
      L     #Abstand;
      CAC;
      -R;
      T     #Abstand;  //Weg für Konstantfahrt
      L     0.0;
      <=R;
      JC    endW;

      L     %DBD14;  //"DI_FW_POS_1".Config.Speed.Norm mm/s
      L     #ProzSpeed;
      *R;
      L     #Abstand;
      CAC;
      /R;
      L     #Warenfahrt;
      +R;
WF:   T     #Warenfahrt;
endW: NOP   0;



NETWORK
TITLE = Hubzeit
      L     #Quelle;
      L     "DB_POS".LENG;
      *D;
      L     "DB_POS".Offset;
      +D;
      SLD   3;
      LAR1;
      OPN   "DB_POS";
      A     DBX [AR1, P#7.6];  //immer schneller Hub
      =     #immer_schnell;

      A     DBX [AR1, P#7.5];  //langsam Heben Badparameter
      O     DBX [AR1, P#38.5];  //WT im Bad
      AN    #immer_schnell;
      =     #lngsm_h;

      L     DBW [AR1, P#84.0];  //Abtropfzeit
      ITD;
      DTR;
      T     #Tropfzeit;

      L     1.0;
      T     #KorrPend;
      T     #KorrAtz;
      SET;
      R     #Trommel;

      L     0;
      L     DBB [AR1, P#36.0];  //WT-DB
      ==I;
      L     0.0;
      JC    Hx;
      CAC;
      +     100;
      T     #WT_DB;

      OPN   DB [#WT_DB];
      L     %DBD38;  //Korrekturfaktor Pendeln
      T     #KorrPend;
      L     %DBD42;  //Korrekturfaktor Abtropfen
      T     #KorrAtz;
      A     %DBX20.0;  //Trommel
      AN    #immer_schnell;
      =     #Trommel;
      A     %DBX22.0;  //langsam senken
      S     #lngsm_s;
      A     %DBX22.1;  //langsam heben
      S     #lngsm_h;

Hx:   L     #Tropfzeit;
      L     #KorrAtz;
      *R;
      T     #Tropfzeit;

      A     #Trommel;
      JC    ATR;
      A     #lngsm_h;
      L     "DB_Fahr-Hubzeit".HZ_Gestell_langsam;
      JC    HZ;
      L     "DB_Fahr-Hubzeit".HZ_Gestell_schnell;
      JU    HZ;

ATR:  A     #lngsm_h;
      L     "DB_Fahr-Hubzeit".HZ_Trommel_langsam;
      JC    HZ;
      L     "DB_Fahr-Hubzeit".HZ_Trommel_schnell;

HZ:   T     #Hubzeit;

NETWORK
TITLE = Senkzeit
      L     #Ziel;
      L     "DB_POS".LENG;
      *D;
      L     "DB_POS".Offset;
      +D;
      SLD   3;
      LAR1;
      OPN   "DB_POS";
      A     DBX [AR1, P#7.6];  //immer schneller Hub
      R     #lngsm_s;
      =     #immer_schnell;

      A     DBX [AR1, P#7.4];  //langsam Senken Badparameter
      AN    #immer_schnell;
      S     #lngsm_s;  //langsam Senken WT-Parameter

      L     DBW [AR1, P#82.0];  //Pendelzeit
      ITD;
      DTR;
      T     #Pendelzeit;
      L     #KorrPend;
      *R;
      T     #Pendelzeit;

      A     #Trommel;
      JC    STR;
      A     #lngsm_s;
      L     "DB_Fahr-Hubzeit".SZ_Gestell_langsam;
      JC    SZ;
      L     "DB_Fahr-Hubzeit".SZ_Gestell_schnell;
      JU    SZ;

STR:  A     #lngsm_s;
      L     "DB_Fahr-Hubzeit".SZ_Trommel_langsam;
      JC    SZ;
      L     "DB_Fahr-Hubzeit".SZ_Trommel_schnell;

SZ:   T     #Senkzeit;

NETWORK
TITLE = Tropfwanne unterschwenken
      AN    #TS_Pos;
      JC    Zeit;
      L     "DB_Fahr-Hubzeit".TS_Zeit;
      L     2.0;
      *R;
      T     #Tropfwanne;

NETWORK
TITLE = Gesamtzeit
Zeit: A     #ChkLeerfahrt;
      L     0.0;
      JC    Korr;
      L     #Restzeit;
      L     #Leerfahrt;
      -R;
      JPZ   Korr;
      L     0.0;
Korr: T     #Restzeit;

      L     #Leerfahrt;
      L     #Restzeit;
      +R;
      L     #Hubzeit;
      +R;
      L     #Tropfzeit;
      +R;
      L     #Tropfwanne;
      +R;
      L     #Warenfahrt;
      +R;
      L     #Pendelzeit;
      +R;
      L     #Senkzeit;
      +R;
      RND+;
      T     #Fahrzeit;

NETWORK
TITLE = Register wiederherstellen
// --------------------------------
// Register wiederherstellen
// --------------------------------
raus: L     #savAr1;
      LAR1;
END_FUNCTION

FUNCTION "FC_VAR_SPL" : Void   // FC13, STL
TITLE = Variable Sprungverteilung
{ S7_Optimized_Access := 'FALSE' }
AUTHOR : MS
// SPRUNGMARKENVORGABE FÜR VARIABLE SCHRITTFOLGEN
// stored: AutoNumber false
   VAR_INPUT
      Instanz_DB : Int;
   END_VAR
   VAR_OUTPUT
      Nr_MicroBef : Byte;
   END_VAR
   VAR_IN_OUT
      next_Step : Bool;
      Adr_MicroBef : Word;
   END_VAR
   VAR_TEMP
      FW_DB : DB_ANY;
      Adresse : DWord;
   END_VAR
BEGIN

NETWORK
TITLE = Programm
// Es ist ab einer festen Adresse des offenen DBs die Reihenfolge der 
// abzuarbeitenden Teilschritte einzugeben. (Schrittnummern der Größe Byte)
      L     #Instanz_DB;
      T     #FW_DB;
      OPN   DI [#FW_DB];

//BEI NEXT WIRD DIE JEWILIGE DB_ADR AKTIVIERT
//DIE SPRUNGADRESSE WIRD ÜBER STEP AUSGEGEBEN
      AN    #next_Step;
      AN    %DIX25.7;  //ZST.Start_UP
      R     %DIX25.2;  //neuer Befehl
      A     %DIX25.7;  //ZST.Start_UP
      JC    Init;
      AN    #next_Step;
      JC    Send;
      L     #Adr_MicroBef;
      L     1;
      +I;
      T     #Adr_MicroBef;
Init: S     %DIX25.2;  //neuer Befehl
      R     %DIX25.3;  //Befehls Merker
      R     %DIX25.4;  //Befehls Merker
      R     %DIX25.5;  //Befehls Merker
      R     %DIX25.6;  //Befehls Merker
      R     %DIX0.4;  //"DI_FW_1".ZST.HEBEN_AKT
      R     %DIX0.5;  //"DI_FW_1".ZST.SENKEN_AKT
      R     %DIX0.6;  //"DI_FW_1".ZST.VORWAERTS_AKT
      R     %DIX0.7;  //"DI_FW_1".ZST.RUECKWAERTS_AKT

Send: L     #Adr_MicroBef;
      SLD   3;
      T     #Adresse;
      L     DIB [#Adresse];
      T     #Nr_MicroBef;
      CLR;
      =     #next_Step;
      =     %DIX25.7;  //ZST.Start_UP
      BE;
END_FUNCTION

FUNCTION "FC_Search_HW" : Void   // FC14, STL
TITLE = ermittelt ggf. HW-Pos
{ S7_Optimized_Access := 'FALSE' }
AUTHOR : MS
// sucht in Fahrtrichtung nach einem notwendigen Höhenwechsel
// und gibt die Höhenwechselposition und die Zielebene zurück
// stored: AutoNumber false
   VAR_INPUT
      SO_li : Bool;   // Sensor Oben aktiv --> kein HW notwendig
      SO_re : Bool;   // Sensor Oben aktiv --> kein HW notwendig
   END_VAR
   VAR_IN_OUT
      IstPos : DInt;   // Istposition des FW in Inkrementen
      ZielPos : DInt;   // Position an der ein Höhenwechsel erfolgt (ohne HW:=tmp.FW_ZIEL_POS)
      Bereich_Ziel : DInt;   // Zielbereich für Positionierung
      Bereich_langsam : DInt;   // Bereich für Langsamfahrt
      FW_Ebene_li : Byte;   // aktuelle FW-Ebene
      Zielebene_li : Byte;   // Ebene die FW im Ziel einnehmen soll
      HW_akt_li : Bool;   // ist dieses Bit gesetzt wurde bereits eine HW-Pos ermittelt
      FW_Ebene_re : Byte;   // aktuelle FW-Ebene
      Zielebene_re : Byte;   // Ebene die FW im Ziel einnehmen soll
      HW_akt_re : Bool;   // ist dieses Bit gesetzt wurde bereits eine HW-Pos ermittelt
   END_VAR
   VAR_TEMP
      count : Int;   // Loopcounter
      fwd : Bool;   // FW bewegt sich in Richtung höhere Position
      HW_Mitte : Bool;   // Höhenwechselposition erreicht
      HW_Pos : DInt;   // an dieser Stelle gilt eine andere Ebene
   END_VAR
BEGIN

NETWORK
TITLE = Initialisierung
// Ist kein Höhenwechsel notwendig wird die aktuelle FW-Ebene als Zielebene und 
// die 
// Tmp.FW_ZIEL_POS als Ziel zurückgegeben.
//Initialisierung
      L     #FW_Ebene_li;
      T     #Zielebene_li;
      L     #FW_Ebene_re;
      T     #Zielebene_re;

      A     #SO_li;
      A     #SO_re;
//existiert ein Höhenwechsel
      ON    "DB_ANLAGE".config.HW_exist;
      R     #HW_akt_li;
      R     #HW_akt_re;
      BEC;

      L     #ZielPos;
      L     #IstPos;
      >D;
      =     #fwd;


NETWORK
TITLE = Scanning
// Suche nach HW-Pos
//FW hat Ziel bereits erreicht
      L     #ZielPos;
      L     #Bereich_Ziel;
      -D;
      L     #IstPos;
      >D;
      JC    chk;
      L     #ZielPos;
      L     #Bereich_Ziel;
      +D;
      L     #IstPos;
      <D;
      JC    chk;
      BE;

chk:  L     0;
retH: T     #count;
      L     "DB_HW".Anzahl;  //HW-Eintrag Länge
      >=I;
      BEC;
      A     #fwd;
      L     #count;
      JC    fwdH;
      +     1;
      -I;
fwdH: L     "DB_HW".lengHW;  //HW-Eintrag Länge
      *I;
      L     "DB_HW".Offset;  //HW-Einträge Offset
      +I;
      SLD   3;
      LAR2;
      OPN   "DB_HW";
      L     0;
      L     DBD [AR2, P#0.0];  //"DB_HW".HW[x].Pos
      ==D;
      BEC;
//HW Mitte?
      L     DBD [AR2, P#0.0];  //"DB_HW".HW[x].Pos
      L     #IstPos;
      -D;
      DTR;
      ABS;
      RND;
      L     #Bereich_Ziel;
      <=D;
      =     #HW_Mitte;
      JC    fnd;

      A     #fwd;
      JC    vor;

//FW hat HW-Pos bereits hinter sich
      L     #IstPos;
      L     DBD [AR2, P#0.0];  //"DB_HW".HW[x].Pos
      <=D;
      JC    nexH;
//Ziel liegt noch vor HW
      L     #ZielPos;
      L     DBD [AR2, P#0.0];  //"DB_HW".HW[x].Pos
      >=D;
      BEC;
//Höhenwechsel liegt auf dem Weg
      JU    fnd;  //Höhenwechel gefunden

vor:  NOP   0;
//FW hat HW-Pos bereits hinter sich
      L     #IstPos;
      L     DBD [AR2, P#0.0];  //"DB_HW".HW[x].Pos
      >=D;
      JC    nexH;
//Ziel liegt noch vor HW
      L     #ZielPos;
      L     DBD [AR2, P#0.0];  //"DB_HW".HW[x].Pos
      <=D;
      BEC;
//Höhenwechsel liegt auf dem Weg
      JU    fnd;  //Höhenwechel gefunden

nexH: L     #count;
      L     1;
      +I;
      JU    retH;

//HW-gefunden
fnd:  A     #SO_li;
      JC    fnd_re;
      A     #fwd;
      JC    fwrd;
      L     DBB [AR2, P#4.0];  //"DB_HW".HW[x].Ebene_rck
      T     #Zielebene_li;
      JU    HWT;
fwrd: L     DBB [AR2, P#5.0];  //"DB_HW".HW[x].Ebene_vor
      T     #Zielebene_li;
HWT:  L     #FW_Ebene_li;
      ==I;
      JC    fnd_re;
      S     #HW_akt_li;
      L     DBD [AR2, P#0.0];  //"DB_HW".HW[x].Pos
      T     #ZielPos;

fnd_re:A     #SO_re;
      BEC;
      A     #fwd;
      JC    fwrd_re;
      L     DBB [AR2, P#4.0];  //"DB_HW".HW[x].Ebene_rck
      T     #Zielebene_re;
      JU    HWT_re;
fwrd_re:L     DBB [AR2, P#5.0];  //"DB_HW".HW[x].Ebene_vor
      T     #Zielebene_re;
HWT_re:L     #FW_Ebene_re;
      ==I;
      BEC;
      S     #HW_akt_re;
      L     DBD [AR2, P#0.0];  //"DB_HW".HW[x].Pos
      T     #ZielPos;
      BE;

END_FUNCTION

FUNCTION "FC_Suche_next_HaltePos" : Void   // FC28, STL
{ S7_Optimized_Access := 'FALSE' }
AUTHOR : MS
// stored: AutoNumber false
   VAR_INPUT
      IstPosInc : DInt;   // IstPos in Inc. (evtl zukünftige Istpos oder Grenzwert)
      Halteweg : DInt;   // Weg zum Anhalten
      vor : Bool;   // Suche in Richtung vorwärts
      SO_li : Bool;   // Zustand oben
      SO_re : Bool;   // Zustand oben
   END_VAR
   VAR_OUTPUT
      ZielPos : Byte;   // nächste mögliche Position zum anhalten
   END_VAR
   VAR_TEMP
      Adr_Reg1 : DWord;   // gerettetes Adreßregister
      Adr_Reg2 : DWord;   // gerettetes Adreßregister
      minPos : Int;
      maxPos : Int;
      ZielInc : DInt;
      IstPos : Int;
      temp_ZielPos : Byte;
   END_VAR
BEGIN

NETWORK
TITLE = Register Sichern
      TAR1;
      T     #Adr_Reg1;
      TAR2;
      T     #Adr_Reg2;


NETWORK
TITLE = 
//-------------------------------------------
//FW-Daten holen
//-------------------------------------------

      L     "DI_FW_1".PAR.Fahrt.FAHRBEREICH_MIN;
      T     #minPos;
      L     "DI_FW_1".PAR.Fahrt.FAHRBEREICH_MAX;
      +     -1;
      T     #maxPos;
      L     "DI_FW_1".ZST.POSITION_li;  // HCA:nur ungerade zählen
      T     #IstPos;
      T     #temp_ZielPos;

//-------------------------------------------
//HalteInkrement bestimmen
//-------------------------------------------
      L     #IstPosInc;
      L     #Halteweg;
      A     #vor;
      JC    add;
      -D;
      JU    stI;
add:  +D;
stI:  T     #ZielInc;

//-------------------------------------------
//Suche HaltePosition
//-------------------------------------------
      L     #temp_ZielPos;
retP: T     #temp_ZielPos;
      L     #minPos;
      <I;
      JC    KorF;
      CAC;
      L     #maxPos;
      >I;
      JC    KorF;

      L     #temp_ZielPos;
      L     "DB_POS".LENG;
      *I;
      L     "DB_POS".Offset;
      +I;
      SLD   3;
      LAR1;
      OPN   "DB_POS";
//Check Dummy-Pos
      L     DBB [AR1, P#0.0];  //Pos-Typ
      L     255;
      ==I;
      JC    nexP;

      L     #temp_ZielPos;
      L     #IstPos;
      <I;
      A     #vor;
      JC    nexP;

      L     #temp_ZielPos;
      L     #IstPos;
      >I;
      AN    #vor;
      JC    nexP;

      L     DBD [AR1, P#22.0];  //Posmitte
      A     #SO_li;
      O     #SO_re;
      JC    nOfs;
      L     DBD [AR1, P#64.0];  //"DB_POS".POS[0].SonderPos_Offset
      -D;
nOfs: L     #ZielInc;
      >=D;
      A     #vor;
      JC    exit;
      <=D;
      AN    #vor;
      JC    exit;

//der nächste bitte
nexP: L     #temp_ZielPos;
      A     #vor;
      +     2;  // HCA nur ungerade zählen
      JC    retP;
      L     #temp_ZielPos;
      +     -2;
      JU    retP;

KorF: T     #temp_ZielPos;
      JU    exit;

NETWORK
TITLE = Register wieder herstellen
exit: L     #Adr_Reg1;
      LAR1;
      L     #Adr_Reg2;
      LAR2;
// Output variablen umkopieren
      L     #temp_ZielPos;
      T     #ZielPos;

END_FUNCTION

FUNCTION "FC_WATCH_SPEED" : Void   // FC15, STL
TITLE = Geschwindigkeitsüberwachung Fahrwagen
{ S7_Optimized_Access := 'FALSE' }
AUTHOR : MS
// Einleitung Soft_Stop bei gefährlicher Annäherung an für die Überfahrt gesperrte 
// Position oder benachbarten Fahrwagen
// Auslösen Not-Stop bei Erreichen bzw. Unterschreitung Mindestabstand
// stored: AutoNumber false
   VAR_INPUT
      Instanz_DB : Int;
      PosInc : DInt;   // Istposition in Inkrementen
      ZielInc : DInt;   // Zielposition in Inkrementen
      Grenze_min : DInt;   // Ende erlaubter Bereich vorwärts
      Grenze_max : DInt;   // Ende erlaubter Bereich rückwärts
      Bereich_lngsm : DInt;   // Bereich für aktivieren der Eilgangverzögerung
      Bereich_Pos : DInt;   // Bereich zur Berechnung der Not-Stop-Adresse
      Dyn_Eil : DInt;   // Bereich für Verzögerung Eilgang
      Offset : Int;   // Offset zur Soft-Stop-Überwachung
      PosGr_min : Bool;   // Minimalgrenzwert durch Bereichsende oder Sperrposition
      PosGr_max : Bool;   // Maximalgrenzwert durch Bereichsende oder Sperrposition
   END_VAR
   VAR_OUTPUT
      PosStop : Bool;   // Position ist Ursache für das Anhalten des FW
      NOTSTOP : Bool;   // Not-Stop an FW
   END_VAR
   VAR_IN_OUT
      Vorwaerts : Bool;   // FW fährt vorwärts
      Rueckwaerts : Bool;   // FW fährt rückwärts
      SoftStop_aktiv : Bool;   // Softstopadresse als Ziel gültig
      ADR_SFT_STOP : DInt;   // POSITION AN DER SOFT-STOP STATT FINDET
   END_VAR
   VAR_TEMP
      FW_DB : DB_ANY;
      ZIEL_FW : DInt;   // ABSTAND ZUM NÄCHSTEN FW IN FAHRTRICHTUNG
      ZIEL_POS : DInt;   // ABSTAND ZUR NÄCHSTEN GESPERRTEN POSITION
      ADR_NOT_STOP : DInt;   // POSITION AN DER NOT-STOP AKTIVIERT WIRD
      Abstand : DInt;   // Abstand zur Soft-Stop-Position
      count : Int;   // Zähler für Suche
      temp_Offset : Int;
      vor : Bool;
      temp_PosStop : Bool;
   END_VAR
BEGIN

NETWORK
TITLE = Initialisieren temporäre Variablen

// Umkopieren der Input Variablen
      L     #Offset;
      T     #temp_Offset;

      L     #Instanz_DB;
      T     #FW_DB;
      OPN   DI [#FW_DB];

//-------------------------------
//RESET TEMPVARIABLE
//-------------------------------
      SET;
      R     #NOTSTOP;
      R     #temp_PosStop;

      A     #Vorwaerts;
      =     #vor;
//-------------------------------
//Abarbeitung nur bei FW_Bewegung
//-------------------------------
      AN    #Vorwaerts;
      AN    #Rueckwaerts;
      JCN   Move;

      A     %DIX12.7;  //"DI_FW_1".ZST.old_vor
      =     #vor;

Move: L     0;
      T     #ZIEL_FW;
      T     #ZIEL_POS;
      T     #ADR_SFT_STOP;
      T     #ADR_NOT_STOP;


NETWORK
TITLE = Annäherung in Fahrtrichtung an Grenzen erlaubter Fahrbereich
// Bereichsgrenzen sind bereits korregiert entsprechend der erlaubten 
// Annäherung.
//-------------------------------
//Richtungserkennung
//-------------------------------
      A     #vor;
      JC    VOR;
//-------------------------------
//Bearbeitung Rückwärtsfahrt
//-------------------------------
      A     #PosGr_min;
      =     #temp_PosStop;
      L     #Grenze_min;  //Ziel Nachbar-FW in Rückwärtsrichtung
      T     #ADR_NOT_STOP;
      JU    CPOS;
//-------------------------------
//Bearbeitung Vorwärtsfahrt
//-------------------------------
VOR:  A     #PosGr_max;
      =     #temp_PosStop;
      L     #Grenze_max;  //Ziel Nachbar-FW in Vorwärtsrichtung
      T     #ADR_NOT_STOP;
//---------------------------
//gesperrte Positon
//---------------------------
CPOS: AN    #temp_PosStop;
      JC    STPS;
      L     0;
      T     #temp_Offset;
//---------------------------
//SoftStop-Position ermitteln
//---------------------------
STPS: L     #Bereich_Pos;
      L     #temp_Offset;
      +D;
      L     #ADR_NOT_STOP;
      CAC;
      A     #vor;
      JC    SUB;
      +D;
      JU    SSTP;
SUB:  -D;
SSTP: T     #ADR_SFT_STOP;


NETWORK
TITLE = Geschwindigkeitskorrektur
// FW setzen auf Langsamfahrt, gezieltes Anhalten und Not-Stop
// Annäherung an Ziel_Pos und Ziel_FW überwachen.
//---------------------
//Not-Stop auslösen
//---------------------
      L     #ZielInc;
      L     #ADR_SFT_STOP;
      A     #vor;
      JC    CVor;
      <D;
      =     #SoftStop_aktiv;
      L     #PosInc;
      L     #ADR_NOT_STOP;
      <D;
      JC    STP;
      JU    Korr;

CVor: >D;
      =     #SoftStop_aktiv;
      L     #PosInc;
      L     #ADR_NOT_STOP;
      >D;
      JC    STP;
      JU    Korr;

//---------------------
//Korrektur notwendig?
//---------------------
Korr: L     #PosInc;
      L     #ADR_SFT_STOP;
      -D;
      DTR;
      ABS;
      RND;
      T     #Abstand;  //Abstand absolut
      JU    Out;  //BE

//-------------------------
//Not-Stop aktiv
//-------------------------
STP:  SET;
      S     #NOTSTOP;
      JU    Out;  //BE

//Umkopieren der Output-Variablen
Out:  A     #temp_PosStop;
      =     #PosStop;
END_FUNCTION

FUNCTION_BLOCK "FB_POS_FW_INC"   // FB21, STL
{ S7_Optimized_Access := 'FALSE' }
AUTHOR : MS
// stored: AutoNumber false
   VAR_INPUT
      SysTime : Time;   // aktuelle Systemzeit
   END_VAR
   VAR
      Config : Struct   // Konfiguration/Einstellungen für Positioniersystem
         Speed : Struct   // Geschwindigkeitsvorgaben
            Min : Int;   // Mindestgeschwindigkeit in %
            Tipp : Int;   // Geschwindigkeit bei Tipp-Betrieb in %
            Hand : Int;   // maximale Geschwindigkeit ohne Freigabe Eil (z.Bsp.:Hand-Betrieb) in %
            Max : Int;   // maximale Geschwindigkeit mit Freigabe Eil (z.Bsp.: Automatik-Betrieb) in %
            Norm : Real;   // Geschwindigkeit in INC/s bei 100%
            endMess : Real;   // gemessene Geschwindigkeit in INC/s bei 100% (wird automatisch ermittelt)
         END_STRUCT;
         Rampe : Struct   // Rampeneinstellungen
            Auf_Leer : Real;   // Zeit für Beschleunigung bei Leerfahrt von 0% auf 200%
            Ab_Leer : Real;   // Zeit für Verzögerung bei Leerfahrt von 200% auf 0%
            Auf_Ware : Real;   // Zeit für Beschleunigung bei Warenfahrt von 0% auf 200%
            Ab_Ware : Real;   // Zeit für Verzögerung bei Warenfahrt von 200% auf 0%
            NotStop : Real;   // Zeit für Verzögerung bei NotStopp von 200% auf 0%
         END_STRUCT;
         Bereich : Struct   // Positionsbereiche
            Pos : DInt;   // gilt als Positionsmitte (nur für Überwachung)
            Stop : DInt;   // Geschwindigkeit==0 Bremse ein
            Ziel : DInt;   // Zielbereich gilt für Ausgabe minSpeed
            Schleich : DInt;   // nur für Sensorsysteme (Schleichgeschwindigkeit)
            Langsam : DInt;   // Bereich der für ein gezieltes Anhalten benötigt wird
         END_STRUCT;
         TV_Position : DInt;   // Verzögerung Positionsmitte in ms
         Reaktionszeit : Int;   // Reaktionszeit FU in ms (Zeit von Ausgabe Sollwert bis Rückmeldung)
         Startzeit : Int;   // Zeit Startverzögerung in ms (Zeit von erster Sollwertausgabe bis Istwert>0)
         Variante : Byte;   // Art der Positionierung (0-Absolut, 1-4SensorSys, 2-..)
         SimIstSpeed : Byte;   // Variante Simulation Istgeschwindigkeit (0-aus, 1-Soll=Ist,...)
         PlateauZeit : Int;   // Zeit[ms] für Plateau zwischen Beschleunigung und Verzögerung
      END_STRUCT;
      IN : Struct   // Eingänge (werden aus FW-DB gelesen (Istwert muß evtl. separat erfasst werden)
         BA_Tipp : Bool;   // Betriebsart FW Tipp
         BA_Hand : Bool;   // Betriebsart FW Hand
         BA_Auto : Bool;   // Betriebsart FW Auto
         LeerFahrt : Bool;   // Leerfahrtparameter verwenden
         Frg_Fahren : Bool;   // Freigabe Positioniervorgang
         Frg_Eil : Bool;   // max. Speed in Automatik und Hand-Speed in Tipp erlaubt
         Break_on : Bool;   // Rückmeldung extern Bremse eingefallen / Wagen steht
         res_2 : Bool;
         resB : Byte;
         PosInc : DInt;   // Istposition in Inkrementen (mm)
         ZielInc : DInt;   // Ziel in Inkrenmenten (mm)
         IstSpeed : Int;   // Istgeschwindigkeit in %
      END_STRUCT;
      OUT : Struct   // Ausgänge werden an FW-DB übergeben (Ausgabe SpeedOut + Umrechnung anlagenspez.)
         Pos_ok : Bool;   // Positionierung beendet FW steht
         Break_off : Bool;   // Bremse lösen
         res_1 : Bool;
         res_2 : Bool;
         res_3 : Bool;
         res_4 : Bool;
         res_5 : Bool;
         res_6 : Bool;
         resB : Byte;
         Bereich_langsam : DInt;   // berechneter Anhaltebereich
         SollSpeed : Int;   // Sollgeschwindigkeit in %
      END_STRUCT;
      Tmp : Struct   // Hilfsvariablen
         lastTime : DInt;   // letzter Systemzeitpunkt
         DiffTime : Real;   // Zeit seit letzter Bearbeitung
         lastSpeed : Real;   // letzte ausgegebene Geschwindigkeit
         Messung : Struct   // Ermittlung der Normgeschwindigkeit
            lastInc : Real;
            addInc : Real;
            addTime : Real;
            lastIst : Int;
            messAct : Bool;
         END_STRUCT;
         StopCount : DInt;   // Zähler für Positionsverzögerung
         subInc : Real;   // Merkzelle für nicht ausgebbare Restwerte
         lastOut : Real;   // im letzten Zyklus ausgegebene Geschwindigkeit
         TaktCount : Real;   // Taktzähler für Sensorsimu
         RunTime : DInt;   // Zeit seit Start Positioniervorgang
      END_STRUCT;
   END_VAR
   VAR_TEMP
      Rampe_Auf : Real;   // aufbereitete Rampe Beschleunigung Dauer in ms bis 100%-Speed
      Rampe_Ab : Real;   // aufbereitete Rampe Verzögerung Dauer in ms von 100% auf 0-Speed
      IstSpeed : Real;   // aufbereitete Istgeschwindigkeit in Inc/ms
      Abstand : Real;   // Abstand zum Ziel (evtl. korrigiert durch Vorhaltezeit)
      minSpeed : Real;   // aktuell geltende Mindestgeschwindigkeit (Regelgrenze)
      maxSpeed : Real;   // aktuell geltende Maximalgeschwindigkeit (Regelgrenze)
      normSpeed : Real;   // Normalgeschwindigkeit bei Sollwert 100% in Inc/ms
      Speed : Real;   // Zwischenergebnis für Ausgabegeschwindigkeit
      maxDelta : Real;   // maximale Änderung der Sollwertvorgabe beim beschleunigen
      messAct : Bool;   // Messung läuf (wird bei 1s konstantem Istwert gesetzt)
      incDelta : DInt;   // zurückgelgter Weg für Ermittlung des NormSpeeds
      Rampe_Not : Real;   // aufbereitete Notrampe (nur in Simulation verwendet)
      Korrmax : Real;   // Korrektur max-Speed vom WT
      HandSpeed : Real;
      TippRampe : Int;
      VOR : Bool;
      RCK : Bool;
      Auto_Befehl : Bool;
      Speicherpos : Bool;
      HandTaste : Bool;
      hiSpeed : Real;   // unkorrigierter max. Speed
      Plateau : Real;
      vPlateau : Real;
      SimSpeed : Bool;
   END_VAR
BEGIN

NETWORK
TITLE = Daten aus FW lesen

      AN    "DI_FW_1".IN.Com_Reset;
      JC    nRes;
      L     #SysTime;
      T     #Tmp.lastTime;
      L     0.0;
      T     #Tmp.lastSpeed;
      T     #Tmp.subInc;

nRes: A     "DI_FW_1".ZST.Auto;
      =     #IN.BA_Auto;
      A     "DI_FW_1".ZST.Hand;
      =     #IN.BA_Hand;
      A     "DI_FW_1".ZST.Tipp;
      O     "DI_FW_1".OUT.TIPP;
      =     #IN.BA_Tipp;
      R     #IN.BA_Auto;
      R     #IN.BA_Hand;

      AN    "DI_FW_1".ZST.Oben_li;
      AN    "DI_FW_1".ZST.Oben_re;
      =     #IN.LeerFahrt;

      A     "DI_FW_1".ZST.MicM2;  //-->Handbetr.Taste gedrückt
      A     #IN.BA_Hand;
      =     #HandTaste;

      A     "DI_FW_1".OUT.VOR;
      =     #VOR;
      A     "DI_FW_1".OUT.RUECK;
      =     #RCK;

      A     #VOR;
      O     #RCK;
      =     #IN.Frg_Fahren;

      A     "DI_FW_1".OUT.POS_EIL;
      =     #IN.Frg_Eil;

      L     "DI_FW_1".ZST.PosInc;
      T     #IN.PosInc;
      L     "DI_FW_1".TMP.FahrZielInc;
      T     #IN.ZielInc;

      CLR;
      =     #Speicherpos;

      L     "DI_FW_1".PAR.Fahrt.WT_Speed;
      ITD;
      DTR;
      L     100.0;
      /R;
      T     #Korrmax;

      L     3;
      L     "DI_FW_1".ZST.BEFEHL.%B2;
      ==I;
      O(;
      L     1;
      ==I;
      );
      =     #Auto_Befehl;

NETWORK
TITLE = kein Auftrag/Initialisieren
//----------------------------------------
//Zeitmessung
//----------------------------------------
      L     #SysTime;
      L     #Tmp.lastTime;
      >=D;
      JC    nUms;
      L     16#7FFF_FFFF;  //L#2147483647
      CAC;
      -D;
      L     #SysTime;
      +D;
      JU    Ums;
nUms: -D;
Ums:  DTR;
      T     #Tmp.DiffTime;
      L     10.0;  //Berechnung unter 10ms zu ungenau
      <R;
      BEC;

      L     #SysTime;
      T     #Tmp.lastTime;

//----------------------------------------
//Parametersatz laden
//----------------------------------------
// :::::::::::::::::::::::::::::::::::::::
// Rampen
// :::::::::::::::::::::::::::::::::::::::
      AN    #IN.LeerFahrt;
      O     #IN.BA_Tipp;
      L     #Config.Rampe.Auf_Ware;
      JC    slu;
      L     #Config.Rampe.Auf_Leer;
slu:  L     1000.0;
      *R;
      L     2.0;
      /R;
      T     #Rampe_Auf;

      AN    #IN.LeerFahrt;
      O     #IN.BA_Tipp;
      L     #Config.Rampe.Ab_Ware;
      JC    sld;
      L     #Config.Rampe.Ab_Leer;
sld:  L     1000.0;
      *R;
      L     2.0;
      /R;
      T     #Rampe_Ab;

// :::::::::::::::::::::::::::::::::::::::
// Normalgeschwindigkeit
// :::::::::::::::::::::::::::::::::::::::
      L     #Config.Speed.Norm;
      L     1000.0;
      /R;
      T     #normSpeed;

// :::::::::::::::::::::::::::::::::::::::
// Istgeschwindigkeit
// :::::::::::::::::::::::::::::::::::::::
      L     #IN.IstSpeed;
      ITD;
      DTR;
      ABS;
      L     10000.0;
      /R;
      L     #normSpeed;
      *R;
      T     #IstSpeed;

// :::::::::::::::::::::::::::::::::::::::
// Abstand
// :::::::::::::::::::::::::::::::::::::::
      L     #IN.PosInc;
      L     #IN.ZielInc;
      -D;
      DTR;
      ABS;
      T     #Abstand;

//Korrektur Abstand (Vorhalteweg)um Reaktionszeit auszugleichen
      L     #Config.Reaktionszeit;  //VorhalteWeg=Istspeed * Reaktionszeit
      ITD;  //s = v*t
      DTR;
      L     #IstSpeed;
      *R;
      L     #Abstand;
      CAC;
      -R;
      L     0.0;
      <=R;
      JC    StA;
      CAC;
StA:  T     #Abstand;

// :::::::::::::::::::::::::::::::::::::::
// --- Geschwindigkeiten (Min, Hand, Max)
// :::::::::::::::::::::::::::::::::::::::
      L     #Config.Speed.Tipp;
      A     #IN.BA_Tipp;
      AN    #IN.Frg_Eil;
      JC    min;
      L     #Config.Speed.Hand;
      A     #IN.BA_Tipp;
      A     #IN.Frg_Eil;
      JC    min;
      L     #Config.Speed.Min;
min:  DTR;
      ABS;
      L     100.0;
      /R;
      L     #normSpeed;
      *R;
      T     #minSpeed;

      L     #Config.Speed.Hand;
      A     #IN.BA_Hand;
      AN    #Auto_Befehl;
      O     #IN.BA_Tipp;
      JC    max;
      L     #Config.Speed.Max;

max:  DTR;
      ABS;
      L     100.0;
      /R;
      L     #normSpeed;
      *R;
      L     #Korrmax;
      *R;
      T     #maxSpeed;
      L     #minSpeed;
      >=R;
      JC    okmx;
      T     #maxSpeed;

//----------------------------------------
//kein Auftrag
//----------------------------------------
okmx: AN    #IN.Frg_Fahren;
      JC    Off;

      L     #Tmp.DiffTime;
      L     #Tmp.RunTime;
      +R;
      T     #Tmp.RunTime;

      AN    #IN.BA_Tipp;
      JC    Auto;

NETWORK
TITLE = Tipp
      L     0;
      L     #Config.SimIstSpeed;
      <>I;
      =     #SimSpeed;

      L     100;
      T     #TippRampe;

      L     #Tmp.lastOut;
      L     #maxSpeed;
      >=R;
      A     #IN.Frg_Eil;
      O(;
      A     #SimSpeed;
      A     #IN.Frg_Eil;
      );
      JC    Tout;
      L     #Tmp.lastOut;
      L     #minSpeed;
      >=R;
      O     #SimSpeed;
      AN    #IN.Frg_Eil;
      JC    Tout;

      L     #Tmp.RunTime;
      L     #TippRampe;
      DTR;
      <R;
      L     #Tmp.lastOut;
      JC    Tout;

      L     0.0;
      T     #Tmp.RunTime;

      L     #normSpeed;
      L     100.0;
      /R;
      L     #Tmp.lastOut;
      +R;
      T     #Tmp.lastOut;
      JU    Tout;

Tout: T     #Speed;

      A     #IN.Frg_Fahren;
      JC    outW;

      L     0.0;
      T     #Tmp.RunTime;
      T     #Tmp.lastOut;
      T     #Speed;

      JU    outW;

NETWORK
TITLE = Positioniervariante aussuchen
Auto: SET;
      R     #OUT.Pos_ok;

      L     #Config.Variante;
      JL    vErr;
      JU    vAbs;  //0 Absolut direkt
      JU    v4FX;  //1 mit 4-Sensor-System
vErr: JU    Off;


NETWORK
TITLE = Positionierung Absolut direkt
vAbs: NOP   0;

//----------------------------------------
// Bereich_Langsam berechnen
//
// s = (Rampe * Vist * Vist) / (2 * Vnorm)
//----------------------------------------
      L     #Rampe_Ab;
      L     0.0;
      <=R;
      L     #Config.Bereich.Langsam;
      JC    setB;

      L     #IstSpeed;
      SQR;
      L     #Rampe_Ab;
      *R;
      L     #normSpeed;
      /R;
      L     2.0;
      /R;
      RND;
setB: T     #OUT.Bereich_langsam;

//----------------------------------------
// maximal mögl. Geschwindigkeit berechnen
//
// v = SQRT(2 * s * Vnorm / Rampe)
//----------------------------------------
      L     #Abstand;
      L     #Config.Bereich.Ziel;
      DTR;
      >R;
      JC    Sped;

      L     #Abstand;
      L     #Config.Bereich.Stop;
      DTR;
      >R;
      L     #minSpeed;
      JC    setS;

      L     0;
      JU    setS;

Sped: L     #Rampe_Ab;
      L     0.0;
      <=R;
      L     #maxSpeed;
      JC    setS;

      L     2.0;
      L     #Abstand;
      *R;
      L     #normSpeed;
      *R;
      L     #Rampe_Ab;
      /R;
      SQRT;
setS: T     #Speed;
      T     #hiSpeed;

//----------------------------------------
// errechnete Geschwindigkeit auf MAX begrenzen
//----------------------------------------
      L     #Speed;
      L     #maxSpeed;
      <=R;
      JC    Ramp;
      T     #Speed;
      JU    Ramp;

//----------------------------------------
// Anstiegsrampe begrenzen
//
// Vdelta = (Vnorm * Tdelta / Rampe)
//----------------------------------------
Ramp: L     #Speed;
      L     #IstSpeed;
      <=R;
      JC    aMin;

      L     #Rampe_Auf;
      L     0.0;
      <=R;
      JC    aMin;

      L     0;
      L     #Config.SimIstSpeed;
      <>I;
      JC    wait;

      L     #IstSpeed;
      L     2.0;
      *R;
      L     #Tmp.lastOut;
      >=R;
      JC    wtr;

wait: L     #Tmp.RunTime;
      L     #Config.Startzeit;
      DTR;
      <R;
      L     #Tmp.lastOut;
      JC    altw;

      L     0;
      L     #Config.SimIstSpeed;
      <>I;
      JC    wtr;

      L     0.0;
      T     #Tmp.RunTime;

      L     #normSpeed;
      L     100.0;
      /R;
      L     #Tmp.lastOut;
      +R;
      T     #Tmp.lastOut;
      JU    altw;

wtr:  L     #normSpeed;
      L     #Tmp.DiffTime;
      *R;
      L     #Rampe_Auf;
      /R;
      T     #maxDelta;

      A     #HandTaste;
      JC    okD;

      L     #Config.PlateauZeit;
      ITD;
      DTR;
      T     #Plateau;

      L     #normSpeed;
      L     #Plateau;  //PlateauZeit
      *R;
      L     #Rampe_Auf;
      /R;
      T     #Plateau;  //Plateau v-Diff

      L     #Plateau;  //Plateau v-Diff
      L     #Tmp.lastOut;
      +R;
      T     #vPlateau;  //PlateauGeschwindigkeit

      L     #hiSpeed;
      L     #vPlateau;
      <=R;
      L     #Tmp.lastOut;
      JC    altw;

      L     #hiSpeed;
      L     #vPlateau;
      -R;
      L     #maxDelta;
      >R;
      JC    okD;
      CAC;
      T     #maxDelta;

okD:  L     #Speed;
      L     #Tmp.lastOut;
      -R;
      ABS;
      L     #maxDelta;
      <=R;
      JC    aMin;

      L     #maxDelta;
      L     #Tmp.lastOut;
      +R;
altw: T     #Speed;

//----------------------------------------
// errechnete Geschwindigkeit auf MIN begrenzen
//----------------------------------------
aMin: L     #Speed;
      L     #minSpeed;
      >=R;
      JC    Out;

      T     #Speed;

      JU    Out;


NETWORK
TITLE = Positionierung mit 4-Sensor-System
v4FX: L     #Config.Speed.Hand;
      ITD;
      DTR;
      L     100.0;
      /R;
      L     #normSpeed;
      *R;
      T     #HandSpeed;

//  L     #Config.Bereich.Langsam
      L     4;
      T     #OUT.Bereich_langsam;

//Schleichen
      L     #Abstand;
      RND;
      L     #Config.Bereich.Schleich;
      <=D;
      L     #minSpeed;
      JC    StFX;

//Langsam
      L     #Config.Bereich.Langsam;
      AN    #Speicherpos;
      JC    Nnor;
      L     #Config.Bereich.Langsam;
      +D;
Nnor: L     #Abstand;
      RND;
      >=D;
      L     #HandSpeed;
      JC    StFX;

//Eil
      L     #maxSpeed;
StFX: T     #Speed;
      JU    Out;


NETWORK
TITLE = Ausgabe
Out:  L     #IN.PosInc;
      L     #IN.ZielInc;
      -D;
      DTR;
      ABS;
      T     #Abstand;

      L     #Config.Variante;
      L     0;
      ==I;
      A(;
      L     #Abstand;
      L     #Config.Bereich.Stop;
      DTR;
      <=R;
      );
      JC    Off;

      L     #IN.ZielInc;
      L     #IN.PosInc;
      -D;
      L     0;
      >D;
      A     #RCK;
      O(;
      <D;
      A     #VOR;
      );
      JC    Off;

      L     #Abstand;
      L     #Config.Bereich.Ziel;
      DTR;
      <=R;
      JC    GOO;

      L     #Config.Variante;
      L     0;
      ==I;
      O     #VOR;
      L     #Config.TV_Position;
      DTR;
      JC    setT;
      L     #Config.Reaktionszeit;
      DTR;
      JU    setT;

GOO:  L     0.0;
      L     #Tmp.StopCount;
      >=R;
      JC    Off;

      L     #Tmp.DiffTime;
      -R;
setT: T     #Tmp.StopCount;
      JU    outW;


Off:  A     #IN.Break_on;
      S     #OUT.Pos_ok;

      L     0;
      T     #OUT.Bereich_langsam;
      L     0.0;
      T     #Speed;
      T     #Tmp.lastOut;
      T     #Tmp.RunTime;
      JU    outW;

outW: L     #Speed;
      T     #Tmp.lastOut;
      L     10000.0;
      *R;
      L     #normSpeed;
      /R;
      T     #maxDelta;
      TRUNC;
      T     #OUT.SollSpeed;

      L     #Tmp.RunTime;
      L     #Config.Startzeit;
      DTR;
      >=R;
      A     #IN.Frg_Fahren;
      S     #OUT.Break_off;

      L     #OUT.SollSpeed;
      L     0;
      ==I;
      ON    #IN.Frg_Fahren;
      R     #OUT.Break_off;


NETWORK
TITLE = Messung der Normgeschwindigkeit
      L     #IN.IstSpeed;
      L     #Tmp.Messung.lastIst;
      -I;
      JP    cNeg;
      NEGI;
cNeg: L     100;
      <=I;
      A     #IN.Frg_Fahren;
      =     #messAct;
      JC    cOn;
//----------------------------------------
// Messung aus
// Werte initialisieren
//----------------------------------------
      L     0.0;
      T     #Tmp.Messung.addTime;
      T     #Tmp.Messung.addInc;

      L     #IN.IstSpeed;
      T     #Tmp.Messung.lastIst;
      JU    cEnd;

//----------------------------------------
// Messung läuft
// Werte aufzeichnen
//----------------------------------------
cOn:  L     #IN.PosInc;
      DTR;
      L     #Tmp.Messung.lastInc;
      -R;
      ABS;
      L     #Tmp.Messung.addInc;
      +R;
      T     #Tmp.Messung.addInc;

      L     #Tmp.DiffTime;
      L     #Tmp.Messung.addTime;
      +R;
      T     #Tmp.Messung.addTime;

//----------------------------------------
// Messung läuft lange genug
// um Werte zu berechnen
//----------------------------------------
      L     #Tmp.Messung.addTime;
      L     1000.0;
      <R;
      JC    cEnd;
      /R;
      L     #Tmp.Messung.addInc;
      CAC;
      /R;
      L     #Tmp.Messung.lastIst;
      ITD;
      DTR;
      ABS;
      /R;
      L     10000.0;
      *R;
      T     #Config.Speed.endMess;
      JU    cEnd;

cEnd: L     #IN.PosInc;
      DTR;
      T     #Tmp.Messung.lastInc;


NETWORK
TITLE = Daten in FW schreiben

      A     #OUT.Pos_ok;
      =     "DI_FW_1".IN.Pos_ok;

      L     #OUT.Bereich_langsam;
      T     "DI_FW_1".PAR.Fahrt.Bereich_lngsm;

      L     #Config.Bereich.Ziel;
      T     "DI_FW_1".PAR.Fahrt.Bereich_Ziel;

      L     #Config.Bereich.Pos;
      T     "DI_FW_1".PAR.Fahrt.Bereich_Pos;

      L     #OUT.SollSpeed;
      T     "DI_FW_1".ZST.Speed_Fahrt;

      L     #Config.Variante;
      L     0;
      <>I;
      L     #Config.Bereich.Langsam;
      JC    setL;

      L     #Config.Reaktionszeit;  //VorhalteWeg=Istspeed * Reaktionszeit
      ITD;  //s = v*t
      DTR;
      L     #maxSpeed;
      *R;
      T     #Abstand;

      L     #maxSpeed;
      SQR;
      L     #Rampe_Ab;
      *R;
      L     #normSpeed;
      /R;
      L     2.0;
      /R;
      L     #Abstand;
      +R;
      RND+;
setL: T     "DI_FW_1".PAR.Fahrt.max_Anhalteweg;


NETWORK
TITLE = Simulation Ist-Wert-Rückgabe
      L     #Config.SimIstSpeed;
      L     0;
      ==I;
      JC    simu;

      L     #OUT.SollSpeed;
      T     #IN.IstSpeed;

      AN    #OUT.Break_off;
      =     #IN.Break_on;

//    BE

simu: NOP   0;

NETWORK
TITLE = Simulation Bewegung
      AN    "DB_ANLAGE".BA.Simulation;
      BEC;

      AN    #OUT.Break_off;
      =     #IN.Break_on;

      L     #Config.Speed.Norm;
      L     1000.0;
      /R;
      T     #normSpeed;

      L     #Config.Rampe.NotStop;
      L     1000.0;
      *R;
      L     2.0;
      /R;
      T     #Rampe_Not;

      L     #normSpeed;
      L     #Tmp.DiffTime;
      *R;
      L     #Rampe_Not;
      /R;
      T     #maxDelta;

      AN    "DI_FW_1".OUT.RUECK;
      JC    sTra;
      L     #Speed;
      NEGR;
      T     #Speed;
sTra: L     #Speed;
      L     #Tmp.lastSpeed;
      -R;
      ABS;
      L     #maxDelta;
      <=R;
      JC    Ink;

      L     #Speed;
      L     #Tmp.lastSpeed;
      <R;
      L     #Tmp.lastSpeed;
      L     #maxDelta;
      JC    sub;
      +R;
      JU    stt;
sub:  -R;
stt:  T     #Speed;

Ink:  L     #Config.Variante;
      JL    sErr;
      JU    sAbs;  //0 Absolut direkt
      JU    sSen;  //1 mit Sensor-System
sErr: JU    OutS;

//----------------------------------------
// Simu Absolut
//----------------------------------------
sAbs: L     #Speed;
      L     #Tmp.lastSpeed;
      +R;
      L     2.0;
      /R;
      L     #Tmp.DiffTime;
      *R;
      L     #Tmp.subInc;
      +R;
      T     #Tmp.subInc;

      TRUNC;
      T     #incDelta;
      L     #IN.PosInc;  // init startinkrement
      +D;
      T     "DI_FW_1".ZST.PosInc;

      L     #Tmp.subInc;
      L     #incDelta;
      DTR;
      -R;
      T     #Tmp.subInc;
      JU    OutS;

//------------------------------------------
// Simu Sensoren
//------------------------------------------
sSen: NOP   0;



      JU    OutS;

//----------------------------------------
// Ausgabe Geschwindigkeit
//----------------------------------------
OutS: L     #Speed;
      T     #Tmp.lastSpeed;


      L     #Config.SimIstSpeed;
      L     0;
      <>I;
      BEC;

      L     #Tmp.lastSpeed;
      L     10000.0;
      *R;
      L     #normSpeed;
      /R;
      ABS;
      TRUNC;
      T     #IN.IstSpeed;

END_FUNCTION_BLOCK

FUNCTION_BLOCK "FB_HUB_FW_li"   // FB22, STL
{ S7_Optimized_Access := 'FALSE' }
AUTHOR : MS
// stored: AutoNumber false
   VAR_INPUT
      FW_DBNr : Int;
      SysTime : Time;
   END_VAR
   VAR
      Config : Struct
         Speed : Struct
            Min : Int;   // Mindestgeschwindigkeit in %
            Tipp : Int;   // Geschwindigkeit bei Tipp-Betrieb in %
            Hand : Int;   // maximale Geschwindigkeit bei Hand-Betrieb in %
            Max : Int;   // maximale Geschwindigkeit bei Automatik-Betrieb in %
            Norm : Real;   // Geschwindigkeit in INC/s bei 100%
            endMess : Real;   // gemessene Geschwindigkeit in INC/s bei 100%
         END_STRUCT;
         Rampe : Struct
            Auf_Heben : Real;   // Zeit für Beschleunigung beim Heben von 0% auf 200%
            Ab_Heben : Real;   // Zeit für Verzögerung bei Heben von 200% auf 0%
            Auf_Senken : Real;   // Zeit für Beschleunigung bei Senken von 0% auf 200%
            Ab_Senken : Real;   // Zeit für Verzögerung bei Senken von 200% auf 0%
            NotStop : Real;   // Zeit für Verzögerung bei NotStopp von 200% auf 0%
         END_STRUCT;
         Bereich : Struct
            Pos : DInt;
            Stop : DInt;
            Ziel : DInt;
            Absetzen : DInt;
            Langsam : DInt;
         END_STRUCT;
         TV_Position : DInt;   // Verzögerung Ebenenmitte in ms
         Reaktionszeit : Int;   // Reaktionszeit FU
         Startzeit : Int;   // Zeit Startverzögerung in ms (Zeit von erster Sollwertausgabe bis Istwert>0)
         Variante : Byte;   // Art der Positionierung (0-Absolut, 1-SensorSys, 2-..)
         SimIstSpeed : Byte;   // Variante Simulation Istgeschwindigkeit (0-aus, 1-Soll=Ist,...)
         SimSensors : DWord := DWORD#16#4400_0022;   // Sensoraufbau für Simulation
         SimTakt : DInt;   // Schiebetakt für Sensorsimu in ms
      END_STRUCT;
      IN : Struct
         BA_Tipp : Bool;   // Betriebsart FW Tipp
         BA_Hand : Bool;   // Betriebsart FW Hand
         BA_Auto : Bool;   // Betriebsart FW Auto
         Heben_aktiv : Bool;
         Frg_Hub : Bool;   // Freigabe Positioniervorgang
         Frg_Eil : Bool;   // max. Speed in Automatik und Hand-Speed in Tipp erlaubt
         Break_on : Bool;   // Rückmeldung extern Bremse eingefallen / Hubwerk steht
         mittig : Bool;   // Hub in Posmitte
         resB : Byte;
         HubInc : DInt;   // Istposition in Inkrementen (mm)
         ZielInc : DInt;   // Ziel in Inkrenmenten (mm)
         Absetz_Inc : DInt;   // Inkrement der SU-Ebene des FW
         IstSpeed : Int;   // Istgeschwindigkeit in %
      END_STRUCT;
      OUT : Struct
         Hub_Ok : Bool;   // Positionierung beendet FW steht
         Break_off : Bool;   // Bremse lösen
         res_1 : Bool;
         res_2 : Bool;
         res_3 : Bool;
         res_4 : Bool;
         res_5 : Bool;
         res_6 : Bool;
         resB : Byte;
         Bereich_langsam : DInt;   // berechneter Anhaltebereich
         SollSpeed : Int;   // Sollgeschwindigkeit in %
      END_STRUCT;
      Tmp : Struct
         lastTime : DInt;   // letzter Systemzeitpunkt
         DiffTime : Real;   // Zeit seit letzter Bearbeitung
         lastSpeed : Real;   // letzte ausgegebene Geschwindigkeit
         Messung : Struct
            lastInc : Real;
            addInc : Real;
            addTime : Real;
            lastIst : Int;
            messAct : Bool;
         END_STRUCT;
         StopCount : DInt;
         subInc : Real;
         lastOut : Real;
         TaktCount : Real;   // Taktzähler für Sensorsimu
         PtrSensors : DWord := DWORD#16#0000_0001;
         RunTime : DInt;   // Zeit seit Start Positioniervorgang
      END_STRUCT;
   END_VAR
   VAR_TEMP
      FWDB : Int;
      Rampe_Auf : Real;
      Rampe_Ab : Real;
      minSpeed : Real;
      maxSpeed : Real;
      normSpeed : Real;
      handSpeed : Real;
      TippSpeed : Real;
      IstSpeed : Real;
      Abstand : Real;
      maxDelta : Real;
      Speed : Real;
      tx : Real;
      Rampe_Not : Real;
      incDelta : DInt;
      messAct : Bool;
      posAbsolut : Bool;
      Sensor_on : Bool;
      no_Brms : Bool;
      savD_1 : DInt;
      savD_2 : DInt;
      Korrmax : Real;   // Korrektur max-Speed vom WT
   END_VAR
BEGIN

NETWORK
TITLE = Daten aus FW lesen

      L     #FW_DBNr;
      T     #FWDB;
      OPN   DB [#FWDB];
      AN    "DI_FW_1".IN.Com_Reset;
      JC    nRes;
      L     #SysTime;
      T     #Tmp.lastTime;
      L     0.0;
      T     #Tmp.lastSpeed;
      T     #Tmp.subInc;

nRes: A     "DI_FW_1".ZST.Auto;
      =     #IN.BA_Auto;
      A     "DI_FW_1".ZST.Hand;
      =     #IN.BA_Hand;
      A     "DI_FW_1".ZST.Tipp;
      O     "DI_FW_1".OUT.TIPP;
      =     #IN.BA_Tipp;
      R     #IN.BA_Auto;
      R     #IN.BA_Hand;

      A     "DI_FW_1".OUT.HEBEN_li;
      =     #IN.Heben_aktiv;

      A     "DI_FW_1".OUT.HEBEN_li;
      O     "DI_FW_1".OUT.SENKEN_li;
      =     #IN.Frg_Hub;

      A     "DI_FW_1".OUT.HUB_EIL_li;
      =     #IN.Frg_Eil;

      A     "DI_FW_1".ZST.Mittig;
      =     #IN.mittig;

      A     "DI_FW_1".OUT.no_Brms;
      =     #no_Brms;

      L     "DI_FW_1".ZST.HubInc_li;
      T     #IN.HubInc;
      L     "DI_FW_1".TMP.HubZielInc_li;
      T     #IN.ZielInc;

      L     "DI_FW_1".TMP.low_SU_Ebene;
      L     4;
      *D;
      L     292;
      +D;
      SLD   3;
      LAR1;
      OPN   DB [#FWDB];
      L     DBD [AR1, P#0.0];  //"DI_FW_1".PAR.Hub.Ebene0
      L     #Config.Bereich.Absetzen;
      +D;
      T     #IN.Absetz_Inc;

      L     "DI_FW_1".PAR.Hub.WT_Speed;
      ITD;
      DTR;
      L     100.0;
      /R;
      L     #Config.Speed.Max;
      ITD;
      DTR;
      *R;
      T     #Korrmax;


NETWORK
TITLE = kein Auftrag/Initialisieren
//----------------------------------------
//Positionierart
//----------------------------------------
      L     #Config.Variante;
      L     0;
      ==I;
      =     #posAbsolut;

//----------------------------------------
//Zeitmessung
//----------------------------------------
      L     #SysTime;
      L     #Tmp.lastTime;
      >=D;
      JC    nUms;
      L     16#7FFF_FFFF;  //L#2147483647
      CAC;
      -D;
      L     #SysTime;
      +D;
      JU    Ums;
nUms: -D;
Ums:  DTR;
      T     #Tmp.DiffTime;
      L     10.0;  //Berechnung unter 10ms zu ungenau
      <R;
      BEC;

      L     #SysTime;
      T     #Tmp.lastTime;

//----------------------------------------
//Parametersatz laden
//----------------------------------------
// :::::::::::::::::::::::::::::::::::::::
// Rampen
// :::::::::::::::::::::::::::::::::::::::
      A     #IN.Heben_aktiv;
      O     #IN.BA_Tipp;
      L     #Config.Rampe.Auf_Heben;
      JC    slu;
      L     #Config.Rampe.Auf_Senken;
slu:  L     1000.0;
      *R;
      L     2.0;
      /R;
      T     #Rampe_Auf;

      A     #IN.Heben_aktiv;
      O     #IN.BA_Tipp;
      L     #Config.Rampe.Ab_Heben;
      JC    sld;
      L     #Config.Rampe.Ab_Senken;
sld:  L     1000.0;
      *R;
      L     2.0;
      /R;
      T     #Rampe_Ab;

// :::::::::::::::::::::::::::::::::::::::
// Normalgeschwindigkeit
// :::::::::::::::::::::::::::::::::::::::
      L     #Config.Speed.Norm;
      L     1000.0;
      /R;
      T     #normSpeed;

// :::::::::::::::::::::::::::::::::::::::
// Istgeschwindigkeit
// :::::::::::::::::::::::::::::::::::::::
      L     #IN.IstSpeed;
      ITD;
      DTR;
      ABS;
      L     10000.0;
      /R;
      L     #normSpeed;
      *R;
      T     #IstSpeed;

// :::::::::::::::::::::::::::::::::::::::
// Abstand
// :::::::::::::::::::::::::::::::::::::::
      L     #IN.HubInc;
      L     #IN.ZielInc;
      -D;
      DTR;
      ABS;
      T     #Abstand;

//Korrektur Abstand (Vorhalteweg)um Reaktionszeit auszugleichen
      AN    #posAbsolut;
      JC    StA;
      L     #Config.Reaktionszeit;  //VorhalteWeg=Istspeed * Reaktionszeit
      ITD;  //s = v*t
      DTR;
      L     #IstSpeed;
      *R;
      L     #Abstand;
      CAC;
      -R;
      L     0.0;
      <=R;
      JC    StA;
      CAC;
StA:  T     #Abstand;


// :::::::::::::::::::::::::::::::::::::::
// --- Geschwindigkeiten (Min, Hand, Max)
// :::::::::::::::::::::::::::::::::::::::
      L     #Config.Speed.Tipp;
      A     #IN.BA_Tipp;
      JC    min;
      L     #Config.Speed.Min;
min:  DTR;
      ABS;
      L     100.0;
      /R;
      L     #normSpeed;
      *R;
      T     #minSpeed;

      L     #Config.Speed.Hand;
      DTR;
      ABS;
      L     100.0;
      /R;
      L     #normSpeed;
      *R;
      T     #handSpeed;

      L     #Config.Speed.Tipp;
      DTR;
      ABS;
      L     100.0;
      /R;
      L     #normSpeed;
      *R;
      T     #TippSpeed;

// 2021-07-09 Heben /Senken gleich
      L     #IN.HubInc;
      L     #IN.Absetz_Inc;
      <=D;
      AN    #IN.Frg_Eil;
      A     #IN.mittig;  // Korb am Haken
      O     #IN.BA_Tipp;
      L     #Config.Speed.Tipp;
      JC    max;

      AN    #IN.mittig;
      L     #Config.Speed.Max;  // Höhenwechsel + Freifahren
      JC    max;

      L     #IN.HubInc;
      L     #IN.Absetz_Inc;
      <=D;
      L     #Config.Speed.Hand;
      PUSH;
      +D;
      JC    max;
//

      L     #Config.Speed.Max;
max:  DTR;
      ABS;
      L     #Korrmax;
      >R;
      JC    korr;
      CAC;
korr: L     100.0;
      /R;
      L     #normSpeed;
      *R;
      T     #maxSpeed;
      L     #minSpeed;
      >=R;
      JC    okmx;
      T     #maxSpeed;

//----------------------------------------
//kein Auftrag
//----------------------------------------
okmx: AN    #IN.Frg_Hub;
      JC    Off;

      L     #Tmp.DiffTime;
      L     #Tmp.RunTime;
      +R;
      T     #Tmp.RunTime;

      AN    #IN.BA_Tipp;
      JC    Auto;


NETWORK
TITLE = Tipp
      A     #IN.Frg_Eil;
      L     #maxSpeed;
      JC    Tout;
      L     #minSpeed;
Tout: T     #Speed;
      JU    OutW;

NETWORK
TITLE = Positioniervariante aussuchen
Auto: SET;
      R     #OUT.Hub_Ok;

      L     #Config.Variante;
      JL    vErr;
      JU    vAbs;  //0 Absolut direkt
      JU    vSen;  //1 mit Sensor-System
vErr: JU    Off;


NETWORK
TITLE = Positionierung Absolut direkt
vAbs: NOP   0;

//----------------------------------------
// Bereich_Langsam berechnen
//
// s = (Rampe * Vist * Vist) / (2 * Vnorm)
//----------------------------------------
      L     #Rampe_Ab;
      L     0.0;
      <=R;
      L     #Config.Bereich.Langsam;
      JC    setB;

      L     #IstSpeed;
      SQR;
      L     #Rampe_Ab;
      *R;
      L     #normSpeed;
      /R;
      L     2.0;
      /R;
      RND;
setB: T     #OUT.Bereich_langsam;

//----------------------------------------
// maximal mögl. Geschwindigkeit berechnen
//
// v = SQRT(2 * s * Vnorm / Rampe)
//----------------------------------------
      L     #Abstand;
      L     #Config.Bereich.Ziel;
      DTR;
      >R;
      JC    Sped;

      L     #Abstand;
      L     #Config.Bereich.Stop;
      DTR;
      >R;
      L     #minSpeed;
      JC    setS;

      L     0;
      JU    setS;

Sped: L     #Rampe_Ab;
      L     0.0;
      <=R;
      L     #maxSpeed;
      JC    setS;

      L     2.0;
      L     #Abstand;
      *R;
      L     #normSpeed;
      *R;
      L     #Rampe_Ab;
      /R;
      SQRT;
setS: T     #Speed;

//----------------------------------------
// MAX begrenzen beim Senken (Absetzen)
//
// Vmax = SQRT(2 * Abstand * V100 / t100 + Vhand * Vhand)
//----------------------------------------
      L     #Rampe_Ab;
      L     0.0;
      <=R;
      O     #IN.Heben_aktiv;
      JC    aMax;

      L     #IN.HubInc;
      L     #IN.Absetz_Inc;
      <=D;
      JC    aMax;

      L     #IN.HubInc;
      L     #IN.Absetz_Inc;
      -D;
      DTR;
      L     2.0;
      *R;
      L     #normSpeed;
      *R;
      L     #Rampe_Ab;
      /R;
      L     #handSpeed;
      SQR;
      +R;
      SQRT;
      L     #maxSpeed;
      >R;
      JC    aMax;
      CAC;
      T     #maxSpeed;

//----------------------------------------
// errechnete Geschwindigkeit auf MAX begrenzen
//----------------------------------------
aMax: L     #Speed;
      L     #maxSpeed;
      <=R;
      JC    Ramp;
      T     #Speed;
      JU    Ramp;

//----------------------------------------
// Anstiegsrampe begrenzen
//
// Vdelta = (Vnorm * Tdelta / Rampe)
//----------------------------------------
Ramp: L     #Speed;
      L     #IstSpeed;
      <=R;
      JC    aMin;

      L     #Rampe_Auf;
      L     0.0;
      <=R;
      JC    aMin;

      L     #Tmp.RunTime;
      L     #Config.Startzeit;
      DTR;
      <R;
      L     #minSpeed;
      JC    altw;

      L     #normSpeed;
      L     #Tmp.DiffTime;
      *R;
      L     #Rampe_Auf;
      /R;
      T     #maxDelta;

      L     #Speed;
      L     #Tmp.lastOut;
      -R;
      ABS;
      L     #maxDelta;
      <=R;
      JC    aMin;

      L     #Tmp.lastOut;
      +R;
altw: T     #Speed;

//----------------------------------------
// errechnete Geschwindigkeit auf MIN begrenzen
//----------------------------------------
aMin: L     #Speed;
      L     #minSpeed;
      >=R;
      JC    Out;

      T     #Speed;

      JU    Out;


NETWORK
TITLE = Positionierung mit Sensor-System
vSen: SET;
// -------------------------------
// Geschwindigkeit berechnen
// -------------------------------
      L     #Abstand;
      L     #Config.Bereich.Langsam;
      DTR;
      >R;
      L     #maxSpeed;
      JC    vSet;

      L     #Abstand;
      L     #Config.Bereich.Ziel;
      DTR;
      <=R;
      L     #minSpeed;
      JC    vSet;

      A     #no_Brms;
      L     #maxSpeed;
      JC    vSet;

      L     #handSpeed;
      L     #maxSpeed;
      >R;
      JC    vSet;
      CAC;

vSet: T     #Speed;

// -------------------------------
// Rampen begrenzen
// -------------------------------
      L     #Speed;
      L     #IstSpeed;
      >R;
      JC    rAuf;
      <R;
      JC    rAb;
      JU    Out;

rAuf: L     0.0;
      L     #Rampe_Auf;
      >=R;
      JC    Out;

      L     #Tmp.RunTime;
      L     #Config.Startzeit;
      DTR;
      >=R;
      JC    wtr2;

      L     #minSpeed;
      JU    outS;

wtr2: L     #normSpeed;
      L     #Tmp.DiffTime;
      *R;
      L     #Rampe_Auf;
      /R;
      T     #maxDelta;

      L     #Speed;
      L     #Tmp.lastOut;
      -R;
      ABS;
      L     #maxDelta;
      <=R;
      JC    Out;

      L     #Tmp.lastOut;
      +R;
outS: T     #Speed;
      JU    Out;

rAb:  L     0.0;
      L     #Rampe_Ab;
      >=R;
      JC    Out;

      L     #normSpeed;
      L     #Tmp.DiffTime;
      *R;
      L     #Rampe_Ab;
      /R;
      T     #maxDelta;

      L     #Tmp.lastOut;
      L     #Speed;
      -R;
      ABS;
      L     #maxDelta;
      <=R;
      JC    Out;

      L     #Tmp.lastOut;
      CAC;
      -R;
      T     #Speed;
      JU    Out;


NETWORK
TITLE = Ausgabe
Out:  L     #Abstand;
      L     #Config.Bereich.Ziel;
      DTR;
      >R;
      L     #Config.TV_Position;
      DTR;
      JC    setT;

      L     #minSpeed;
      T     #Speed;

      L     #Tmp.StopCount;
      L     0.0;
      <=R;
      O(;
      L     #Abstand;
      L     #Config.Bereich.Stop;
      DTR;
      <=R;
      A     #posAbsolut;
      );
      JC    Off;

      L     #Tmp.StopCount;
      L     #Tmp.DiffTime;
      -R;

setT: T     #Tmp.StopCount;
      JU    OutW;

Off:  A     #IN.Break_on;
      S     #OUT.Hub_Ok;

      L     0;
      T     #OUT.Bereich_langsam;
      L     0.0;
      T     #Speed;
      T     #Tmp.lastOut;
      T     #Tmp.RunTime;
      JU    OutW;

OutW: L     #Speed;
      T     #Tmp.lastOut;
      L     100.0;
      *R;
      L     #normSpeed;
      /R;
      T     #maxDelta;
      TRUNC;
      T     #OUT.SollSpeed;

      L     #Tmp.RunTime;
      L     #Config.Startzeit;
      DTR;
      >=R;
      A     #IN.Frg_Hub;
      S     #OUT.Break_off;

      L     #OUT.SollSpeed;
      L     0;
      ==I;
      ON    #IN.Frg_Hub;
      R     #OUT.Break_off;


NETWORK
TITLE = Messung der Normgeschwindigkeit
      L     #IN.IstSpeed;
      L     #Tmp.Messung.lastIst;
      -I;
      JP    cNeg;
      NEGI;
cNeg: L     100;
      <=I;
      A     #IN.Frg_Hub;
      =     #messAct;
      JC    cOn;
//----------------------------------------
// Messung aus
// Werte initialisieren
//----------------------------------------
      L     0.0;
      T     #Tmp.Messung.addTime;
      T     #Tmp.Messung.addInc;

      L     #IN.IstSpeed;
      T     #Tmp.Messung.lastIst;
      JU    cEnd;

//----------------------------------------
// Messung läuft
// Werte aufzeichnen
//----------------------------------------
cOn:  L     #IN.HubInc;
      DTR;
      L     #Tmp.Messung.lastInc;
      -R;
      ABS;
      L     #Tmp.Messung.addInc;
      +R;
      T     #Tmp.Messung.addInc;

      L     #Tmp.DiffTime;
      L     #Tmp.Messung.addTime;
      +R;
      T     #Tmp.Messung.addTime;

//----------------------------------------
// Messung läuft lange genug
// um Werte zu berechnen
//----------------------------------------
      L     #Tmp.Messung.addTime;
      L     1000.0;
      <R;
      JC    cEnd;
      /R;
      L     #Tmp.Messung.addInc;
      CAC;
      /R;
      L     #Tmp.Messung.lastIst;
      ITD;
      DTR;
      ABS;
      /R;
      L     10000.0;
      *R;
      T     #Config.Speed.endMess;
      JU    cEnd;

cEnd: L     #IN.HubInc;
      DTR;
      T     #Tmp.Messung.lastInc;



NETWORK
TITLE = Daten in FW schreiben

      OPN   DB [#FWDB];

      A     #OUT.Hub_Ok;
      =     "DI_FW_1".IN.Hub_ok_li;

      L     #OUT.Bereich_langsam;
      T     "DI_FW_1".PAR.Hub.Bereich_lngsm;

      L     #Config.Bereich.Ziel;
      T     "DI_FW_1".PAR.Hub.Bereich_Ziel;

      L     #Config.Bereich.Pos;
      T     "DI_FW_1".PAR.Hub.Bereich_Pos;

      L     #OUT.SollSpeed;
      T     "DI_FW_1".ZST.Speed_Hub_li;


NETWORK
TITLE = Simulation Ist-Wert-Rückgabe
      L     #Config.SimIstSpeed;
      L     0;
      ==I;
      JC    simu;

      L     #OUT.SollSpeed;
      T     #IN.IstSpeed;

simu: NOP   0;


NETWORK
TITLE = Simulation Bewegung
      AN    "DB_ANLAGE".BA.Simulation;
      BEC;

      AN    #OUT.Break_off;
      =     #IN.Break_on;

      A     #IN.Heben_aktiv;
      JC    sTra;
      L     #Speed;
      NEGR;
      T     #Speed;
sTra: L     #Config.Rampe.NotStop;
      L     0.0;
      <=R;
      JC    Ink;

      L     #Config.Rampe.NotStop;
      L     1000.0;
      *R;
      L     2.0;
      /R;
      T     #Rampe_Not;

      L     #normSpeed;
      L     #Tmp.DiffTime;
      *R;
      L     #Rampe_Not;
      /R;
      T     #maxDelta;

      L     #Speed;
      L     #Tmp.lastSpeed;
      -R;
      ABS;
      L     #maxDelta;
      <=R;
      JC    Ink;

      L     #Speed;
      L     #Tmp.lastSpeed;
      <R;
      L     #Tmp.lastSpeed;
      L     #maxDelta;
      JC    sub;
      +R;
      JU    stt;
sub:  -R;
stt:  T     #Speed;

Ink:  L     #Config.Variante;
      JL    sErr;
      JU    sAbs;  //0 Absolut direkt
      JU    sSen;  //1 mit Sensor-System
sErr: JU    OutS_Mig;

//----------------------------------------
// Simu Absolut
//----------------------------------------
sAbs: L     #Speed;
      L     #Tmp.lastSpeed;
      +R;
      L     2.0;
      /R;
      L     #Tmp.DiffTime;
      *R;
      L     #Tmp.subInc;
      +R;
      T     #Tmp.subInc;

      TRUNC;
      T     #incDelta;
      L     #IN.HubInc;  // init startinkrement
      +D;
      OPN   DB [#FWDB];
      T     "DI_FW_1".ZST.HubInc_li;

      L     #Tmp.subInc;
      L     #incDelta;
      DTR;
      -R;
      T     #Tmp.subInc;
      JU    OutS_Mig;

//------------------------------------------
// Simu Sensoren
//------------------------------------------

// :::::::::::::::::::::::::::::::::::::::::
// Simulationstakt entsprechend IstSpeed
// verlängern oder verkürzen
// :::::::::::::::::::::::::::::::::::::::::
sSen: L     #Speed;
      L     #Tmp.lastSpeed;
      +R;
      L     2.0;
      /R;
      ABS;
      L     #normSpeed;
      /R;
      L     #Tmp.DiffTime;
      *R;
      L     #Tmp.TaktCount;
      CAC;
      -R;
      T     #Tmp.TaktCount;

// :::::::::::::::::::::::::::::::::::::::::
// Simutakt abgelaufen --> Pointer schieben
// :::::::::::::::::::::::::::::::::::::::::
      L     0.0;
      L     #Tmp.TaktCount;
      <R;
      ON    #IN.Frg_Hub;
      JC    sInc;
      L     #Config.SimTakt;
      DTR;
      +R;
      T     #Tmp.TaktCount;

      L     0;
      L     #Tmp.PtrSensors;
      ==D;
      JC    UIn;

      L     #Tmp.PtrSensors;  //Pointer (virtuelle Höhe)
      A     #IN.Heben_aktiv;
      JC    hSim;
      SRD   1;  //Pointer (virtuelle Höhe) nach unten
      JP    UIn;  //Unterlauf
      JU    tSim;
hSim: SLD   1;  //Pointer (virtuelle Höhe) nach oben
      JP    OIn;  //Überlauf
tSim: T     #Tmp.PtrSensors;

// :::::::::::::::::::::::::::::::::::::::::
// Istposition ermitteln
// :::::::::::::::::::::::::::::::::::::::::
sInc: L     0;
      T     #incDelta;
      SET;
      R     #Sensor_on;

      L     #Tmp.PtrSensors;  //Zeiger auf virtuelle Höhe
      L     #Config.SimSensors;  //Jedes Bit=1 ist ein Sensor
retR: SRD   1;  //nach Sensoren suchen
      JP    posR;

      A     #Sensor_on;  //Sensor verlassen --> Zählen
      R     #Sensor_on;
      JC    cntR;
      JU    nexR;

posR: AN    #Sensor_on;  //Sensor erreicht --> Zählen
      S     #Sensor_on;
      JC    cntR;
      JU    nexR;

cntR: T     #savD_1;  //Akku 1 retten
      CAC;
      T     #savD_2;  //Akku 2 retten
      L     #incDelta;  //Inkrement erhöhen
      L     1;
      +D;
      T     #incDelta;
      L     #savD_2;  //Akkus wieder herstellen
      L     #savD_1;  //geschobene Werte zur weiterverarbeitung

nexR: CAC;
      SRD   1;  //Pointer schieben
      JP    endR;  //Pointer gefunden --> alle Inkremente gezählt
      CAC;
      JU    retR;  //weiterzählen

endR: L     #incDelta;
      OPN   DB [#FWDB];
      T     %DBD8;  //"DI_FW_1".ZST.HubInc
      JU    OutS_Mig;

UIn:  L     1;  //bei Unterlauf Pointer initialisieren
      T     #Tmp.PtrSensors;
      JU    OutS_Mig;

OIn:  L     16#8000_0000;  //bei Überlauf Pointer initialisieren
      T     #Tmp.PtrSensors;
      JU    OutS_Mig;

//----------------------------------------
// Ausgabe Geschwindigkeit
//----------------------------------------
OutS_Mig:L     #Speed;
      T     #Tmp.lastSpeed;


      L     #Config.SimIstSpeed;
      L     0;
      <>I;
      BEC;

      L     #Tmp.lastSpeed;
      L     10000.0;
      *R;
      L     #normSpeed;
      /R;
      ABS;
      TRUNC;
      T     #IN.IstSpeed;

END_FUNCTION_BLOCK

